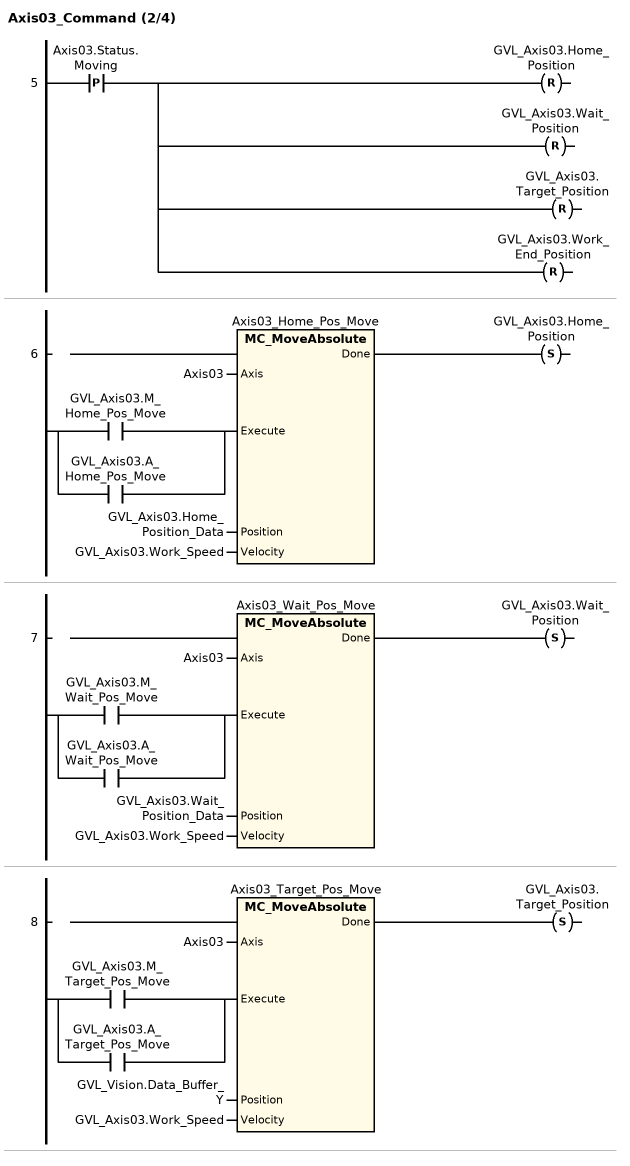
// NETWORK 5
_rt2(CLK := Axis03.Status.Moving);
GVL_Axis03.Home_Position R= _rt2.Q;
GVL_Axis03.Wait_Position R= _rt2.Q;
GVL_Axis03.Target_Position R= _rt2.Q;
GVL_Axis03.Work_End_Position R= _rt2.Q;

// NETWORK 6
Axis03_Home_Pos_Move(
    Axis := Axis03,
    Execute := GVL_Axis03.M_Home_Pos_Move OR GVL_Axis03.A_Home_Pos_Move,
    Position := GVL_Axis03.Home_Position_Data,
    Velocity := GVL_Axis03.Work_Speed); // MC_MoveAbsolute
GVL_Axis03.Home_Position S= Axis03_Home_Pos_Move.Done;

// NETWORK 7
Axis03_Wait_Pos_Move(
    Axis := Axis03,
    Execute := GVL_Axis03.M_Wait_Pos_Move OR GVL_Axis03.A_Wait_Pos_Move,
    Position := GVL_Axis03.Wait_Position_Data,
    Velocity := GVL_Axis03.Work_Speed); // MC_MoveAbsolute
GVL_Axis03.Wait_Position S= Axis03_Wait_Pos_Move.Done;

// NETWORK 8
Axis03_Target_Pos_Move(
    Axis := Axis03,
    Execute := GVL_Axis03.M_Target_Pos_Move OR GVL_Axis03.A_Target_Pos_Move,
    Position := GVL_Vision.Data_Buffer_Y,
    Velocity := GVL_Axis03.Work_Speed); // MC_MoveAbsolute
GVL_Axis03.Target_Position S= Axis03_Target_Pos_Move.Done;

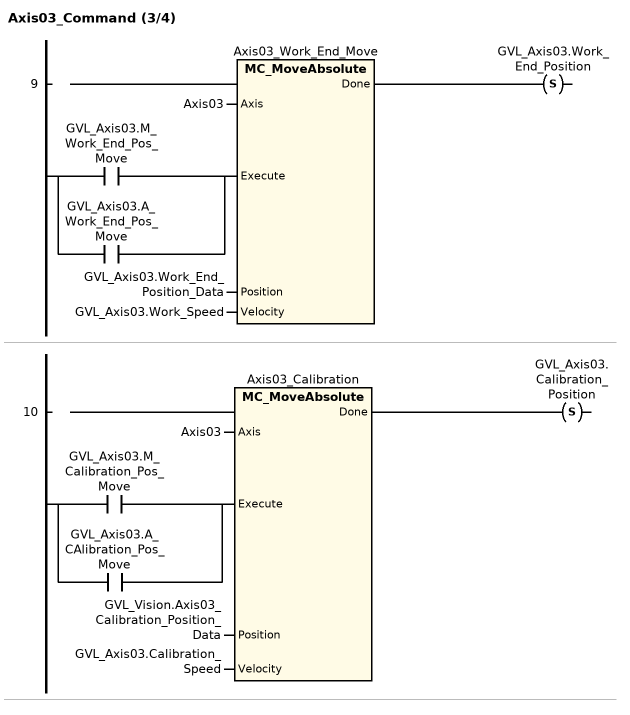
// NETWORK 9
Axis03_Work_End_Move(
    Axis := Axis03,
    Execute := GVL_Axis03.M_Work_End_Pos_Move OR GVL_Axis03.A_Work_End_Pos_Move,
    Position := GVL_Axis03.Work_End_Position_Data,
    Velocity := GVL_Axis03.Work_Speed); // MC_MoveAbsolute
GVL_Axis03.Work_End_Position S= Axis03_Work_End_Move.Done;

// NETWORK 10
Axis03_Calibration(
    Axis := Axis03,
    Execute := GVL_Axis03.M_Calibration_Pos_Move OR GVL_Axis03.A_CAlibration_Pos_Move,
    Position := GVL_Vision.Axis03_Calibration_Position_Data,
    Velocity := GVL_Axis03.Calibration_Speed); // MC_MoveAbsolute
GVL_Axis03.Calibration_Position S= Axis03_Calibration.Done;

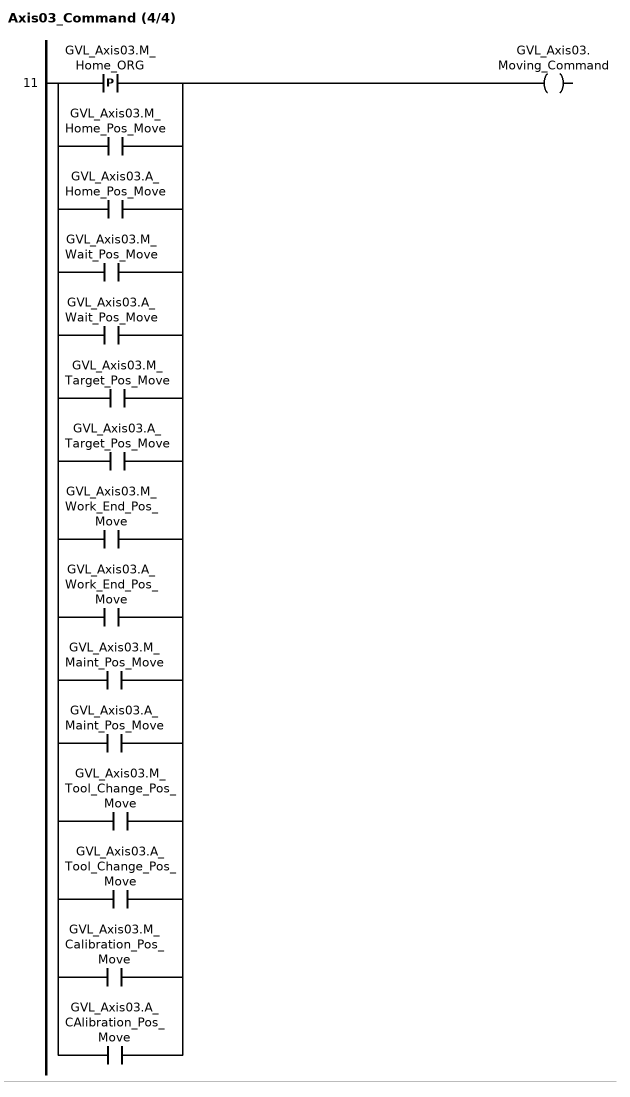
// NETWORK 11
_rt3(CLK := GVL_Axis03.M_Home_ORG);
GVL_Axis03.Moving_Command := _rt3.Q OR GVL_Axis03.M_Home_Pos_Move OR GVL_Axis03.A_Home_Pos_Move OR GVL_Axis03.M_Wait_Pos_Move OR GVL_Axis03.A_Wait_Pos_Move OR GVL_Axis03.M_Target_Pos_Move OR GVL_Axis03.A_Target_Pos_Move OR GVL_Axis03.M_Work_End_Pos_Move OR GVL_Axis03.A_Work_End_Pos_Move OR GVL_Axis03.M_Maint_Pos_Move OR GVL_Axis03.A_Maint_Pos_Move OR GVL_Axis03.M_Tool_Change_Pos_Move OR GVL_Axis03.A_Tool_Change_Pos_Move OR GVL_Axis03.M_Calibration_Pos_Move OR GVL_Axis03.A_CAlibration_Pos_Move;

END_PROGRAM

// ---- POUs/Axis03_Y/Axis03_Manual.TcPOU
PROGRAM Axis03_Manual
VAR
	Always_ON	:	BOOL	:=TRUE	;//상시 ON 
	Always_OFF	:	BOOL	:=FALSE	;//상시 OFF
END_VAR
VAR // added by the converter: edge detectors and wires of the graphical bodies
    _rt1, _rt2, _rt3 : R_TRIG;
END_VAR

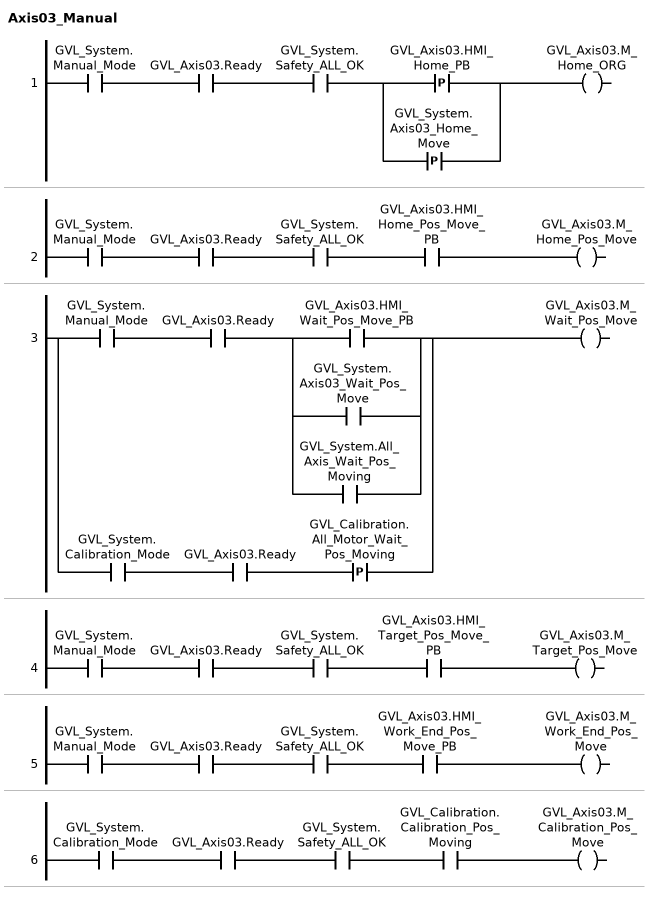
// NETWORK 1
_rt1(CLK := GVL_Axis03.HMI_Home_PB);
_rt2(CLK := GVL_System.Axis03_Home_Move);
GVL_Axis03.M_Home_ORG := GVL_System.Manual_Mode AND GVL_Axis03.Ready AND GVL_System.Safety_ALL_OK AND (_rt1.Q OR _rt2.Q);

// NETWORK 2
GVL_Axis03.M_Home_Pos_Move := GVL_System.Manual_Mode AND GVL_Axis03.Ready AND GVL_System.Safety_ALL_OK AND GVL_Axis03.HMI_Home_Pos_Move_PB;

// NETWORK 3
_rt3(CLK := GVL_Calibration.All_Motor_Wait_Pos_Moving);
GVL_Axis03.M_Wait_Pos_Move := GVL_System.Manual_Mode AND GVL_Axis03.Ready AND (GVL_Axis03.HMI_Wait_Pos_Move_PB OR GVL_System.Axis03_Wait_Pos_Move OR GVL_System.All_Axis_Wait_Pos_Moving) OR GVL_System.Calibration_Mode AND GVL_Axis03.Ready AND _rt3.Q;

// NETWORK 4
GVL_Axis03.M_Target_Pos_Move := GVL_System.Manual_Mode AND GVL_Axis03.Ready AND GVL_System.Safety_ALL_OK AND GVL_Axis03.HMI_Target_Pos_Move_PB;

// NETWORK 5
GVL_Axis03.M_Work_End_Pos_Move := GVL_System.Manual_Mode AND GVL_Axis03.Ready AND GVL_System.Safety_ALL_OK AND GVL_Axis03.HMI_Work_End_Pos_Move_PB;

// NETWORK 6
GVL_Axis03.M_Calibration_Pos_Move := GVL_System.Calibration_Mode AND GVL_Axis03.Ready AND GVL_System.Safety_ALL_OK AND GVL_Calibration.Calibration_Pos_Moving;

END_PROGRAM

// ---- POUs/Axis03_Y/Axis03_Auto.TcPOU
PROGRAM Axis03_Auto
VAR
//System_Bit
	Always_ON	:	BOOL	:=TRUE	;//상시 ON 
	Always_OFF	:	BOOL	:=FALSE	;//상시 OFF
END_VAR

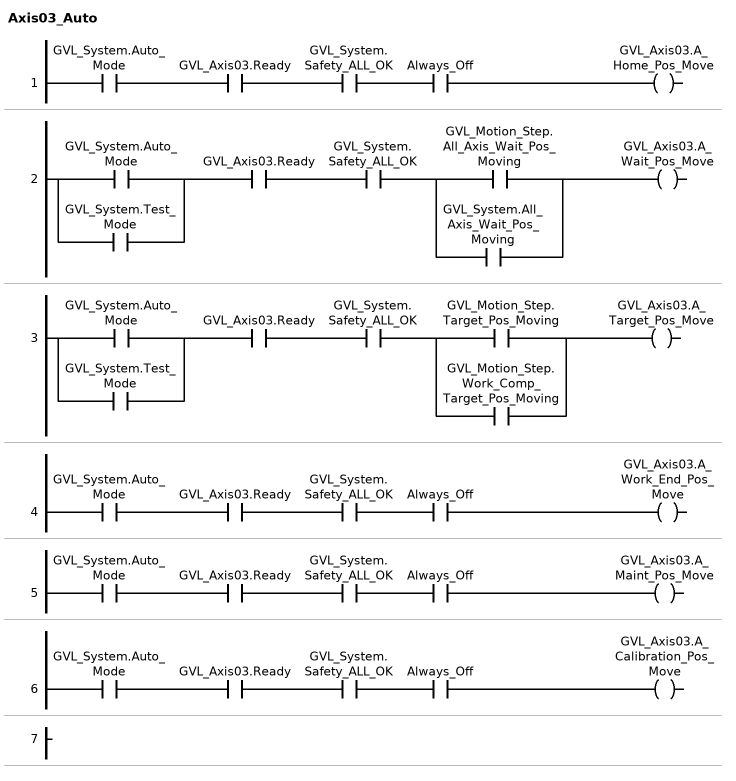
// NETWORK 1
GVL_Axis03.A_Home_Pos_Move := GVL_System.Auto_Mode AND GVL_Axis03.Ready AND GVL_System.Safety_ALL_OK AND Always_Off;

// NETWORK 2
GVL_Axis03.A_Wait_Pos_Move := (GVL_System.Auto_Mode OR GVL_System.Test_Mode) AND GVL_Axis03.Ready AND GVL_System.Safety_ALL_OK AND (GVL_Motion_Step.All_Axis_Wait_Pos_Moving OR GVL_System.All_Axis_Wait_Pos_Moving);

// NETWORK 3
GVL_Axis03.A_Target_Pos_Move := (GVL_System.Auto_Mode OR GVL_System.Test_Mode) AND GVL_Axis03.Ready AND GVL_System.Safety_ALL_OK AND (GVL_Motion_Step.Target_Pos_Moving OR GVL_Motion_Step.Work_Comp_Target_Pos_Moving);

// NETWORK 4
GVL_Axis03.A_Work_End_Pos_Move := GVL_System.Auto_Mode AND GVL_Axis03.Ready AND GVL_System.Safety_ALL_OK AND Always_Off;

// NETWORK 5
GVL_Axis03.A_Maint_Pos_Move := GVL_System.Auto_Mode AND GVL_Axis03.Ready AND GVL_System.Safety_ALL_OK AND Always_Off;

// NETWORK 6
GVL_Axis03.A_Calibration_Pos_Move := GVL_System.Auto_Mode AND GVL_Axis03.Ready AND GVL_System.Safety_ALL_OK AND Always_Off;

// NETWORK 7

END_PROGRAM

// ---- POUs/Axis03_Y/Axis03_Alarm.TcPOU
PROGRAM Axis03_Alarm
VAR
	Always_ON	:	BOOL	:=TRUE	;//상시 ON 
	Always_OFF	:	BOOL	:=FALSE	;//상시 OFF
END_VAR

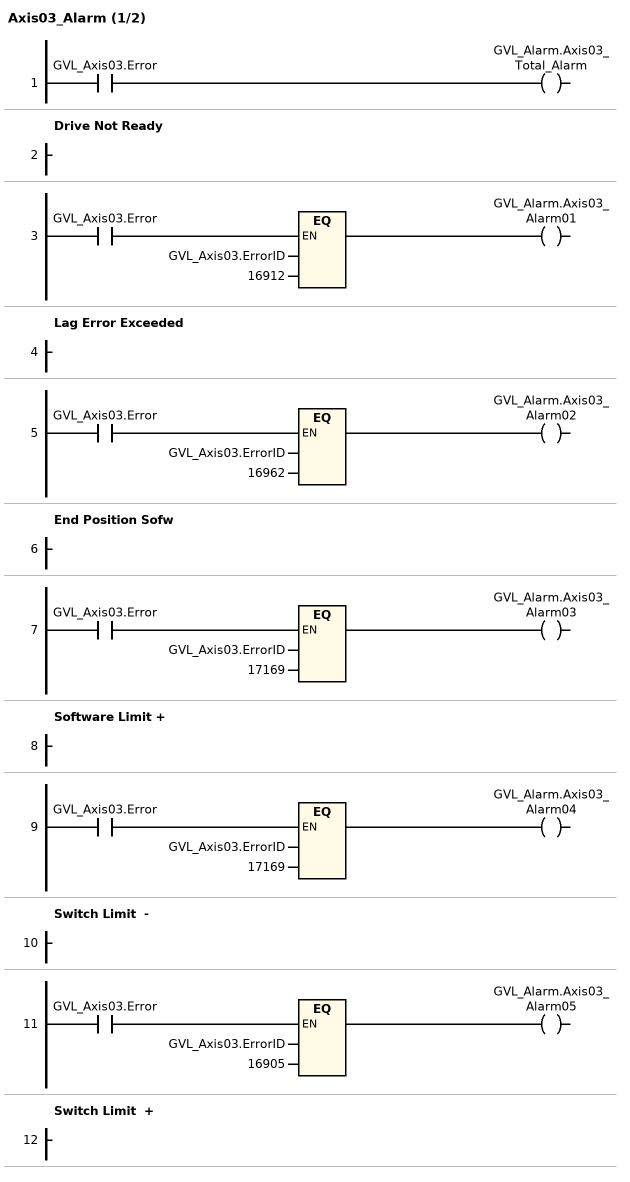
// NETWORK 1
GVL_Alarm.Axis03_Total_Alarm := GVL_Axis03.Error;

// NETWORK 2: Drive Not Ready

// NETWORK 3
GVL_Alarm.Axis03_Alarm01 := GVL_Axis03.Error AND GVL_Axis03.ErrorID = 16912;

// NETWORK 4: Lag Error Exceeded

// NETWORK 5
GVL_Alarm.Axis03_Alarm02 := GVL_Axis03.Error AND GVL_Axis03.ErrorID = 16962;

// NETWORK 6: End Position Sofw

// NETWORK 7
GVL_Alarm.Axis03_Alarm03 := GVL_Axis03.Error AND GVL_Axis03.ErrorID = 17169;

// NETWORK 8: Software Limit +

// NETWORK 9
GVL_Alarm.Axis03_Alarm04 := GVL_Axis03.Error AND GVL_Axis03.ErrorID = 17169;

// NETWORK 10: Switch Limit -

// NETWORK 11
GVL_Alarm.Axis03_Alarm05 := GVL_Axis03.Error AND GVL_Axis03.ErrorID = 16905;

// NETWORK 12: Switch Limit +

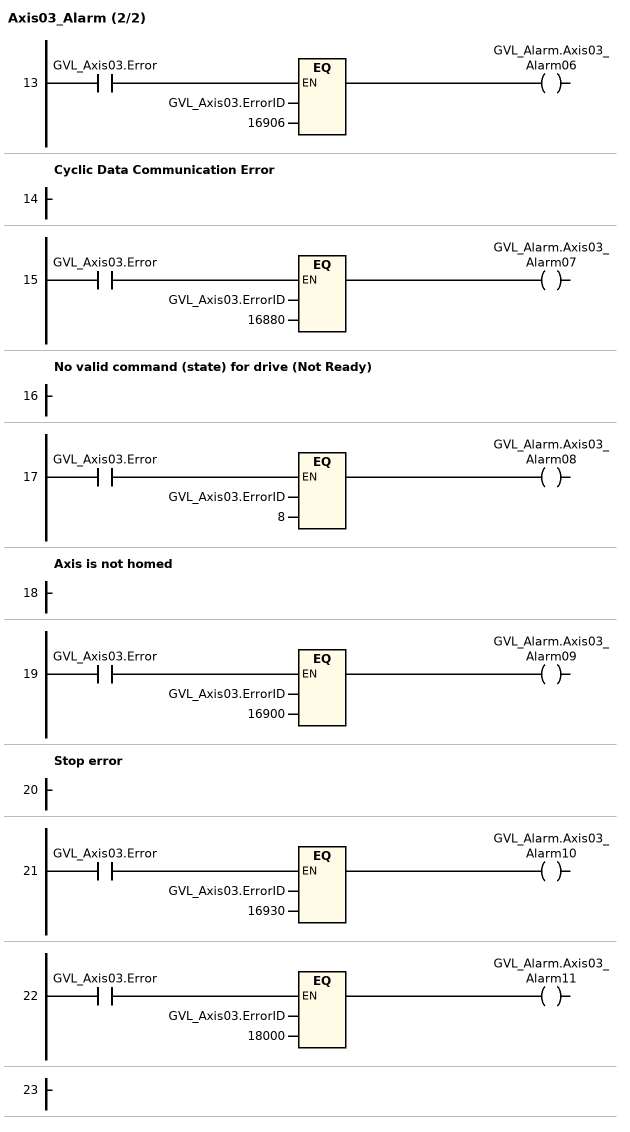
// NETWORK 13
GVL_Alarm.Axis03_Alarm06 := GVL_Axis03.Error AND GVL_Axis03.ErrorID = 16906;

// NETWORK 14: Cyclic Data Communication Error

// NETWORK 15
GVL_Alarm.Axis03_Alarm07 := GVL_Axis03.Error AND GVL_Axis03.ErrorID = 16880;

// NETWORK 16: No valid command (state) for drive (Not Ready)

// NETWORK 17
GVL_Alarm.Axis03_Alarm08 := GVL_Axis03.Error AND GVL_Axis03.ErrorID = 8;

// NETWORK 18: Axis is not homed

// NETWORK 19
GVL_Alarm.Axis03_Alarm09 := GVL_Axis03.Error AND GVL_Axis03.ErrorID = 16900;

// NETWORK 20: Stop error

// NETWORK 21
GVL_Alarm.Axis03_Alarm10 := GVL_Axis03.Error AND GVL_Axis03.ErrorID = 16930;

// NETWORK 22
GVL_Alarm.Axis03_Alarm11 := GVL_Axis03.Error AND GVL_Axis03.ErrorID = 18000;

// NETWORK 23

END_PROGRAM

// ---- POUs/Axis04_Z/Axis04_Status.TcPOU
PROGRAM Axis04_Status
VAR
//System_Bit
	Always_ON	:	BOOL	:=TRUE	;//상시 ON 
	Always_OFF	:	BOOL	:=FALSE	;//상시 OFF
	
//Motor_Command
	Axis04_Status_01: MC_ReadStatus;
	Axis04_Position_Read_01: MC_ReadActualPosition;
	Axis04_Velocity_Read_01: MC_ReadActualVelocity;
	Axis04_Reset_01: MC_Reset;
	Axis04_Stop_01: MC_Stop;
	Torque_Down : UINT := 1500;
	Torque_Up : UINT := 1500;
END_VAR
VAR // added by the converter: edge detectors and wires of the graphical bodies
    _rt1 : R_TRIG;
END_VAR

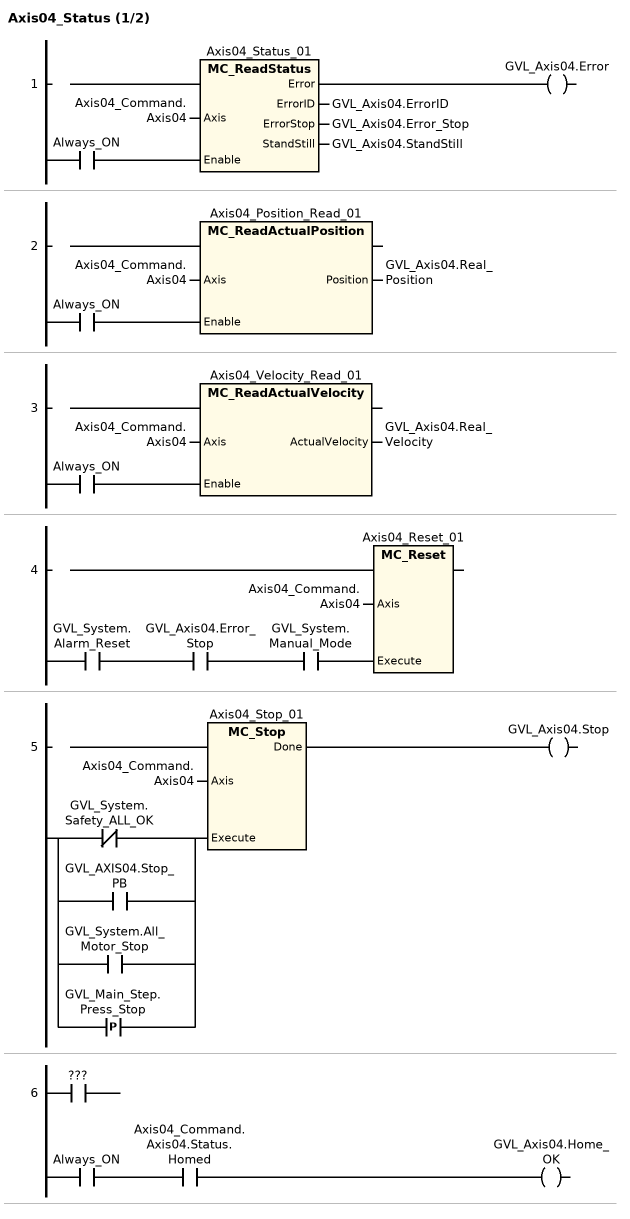
// NETWORK 1
Axis04_Status_01(
    Axis := Axis04_Command.Axis04,
    Enable := Always_ON,
    Error => GVL_Axis04.Error,
    ErrorID => GVL_Axis04.ErrorID,
    ErrorStop => GVL_Axis04.Error_Stop,
    StandStill => GVL_Axis04.StandStill); // MC_ReadStatus

// NETWORK 2
Axis04_Position_Read_01(
    Axis := Axis04_Command.Axis04,
    Enable := Always_ON,
    Position => GVL_Axis04.Real_Position); // MC_ReadActualPosition

// NETWORK 3
Axis04_Velocity_Read_01(
    Axis := Axis04_Command.Axis04,
    Enable := Always_ON,
    ActualVelocity => GVL_Axis04.Real_Velocity); // MC_ReadActualVelocity

// NETWORK 4
Axis04_Reset_01(Axis := Axis04_Command.Axis04, Execute := GVL_System.Alarm_Reset AND GVL_Axis04.Error_Stop AND GVL_System.Manual_Mode); // MC_Reset

// NETWORK 5
_rt1(CLK := GVL_Main_Step.Press_Stop);
Axis04_Stop_01(Axis := Axis04_Command.Axis04, Execute := NOT GVL_System.Safety_ALL_OK OR GVL_AXIS04.Stop_PB OR GVL_System.All_Motor_Stop OR _rt1.Q); // MC_Stop
GVL_Axis04.Stop := Axis04_Stop_01.Done;

// NETWORK 6
GVL_Axis04.Home_OK := Always_ON AND Axis04_Command.Axis04.Status.Homed;

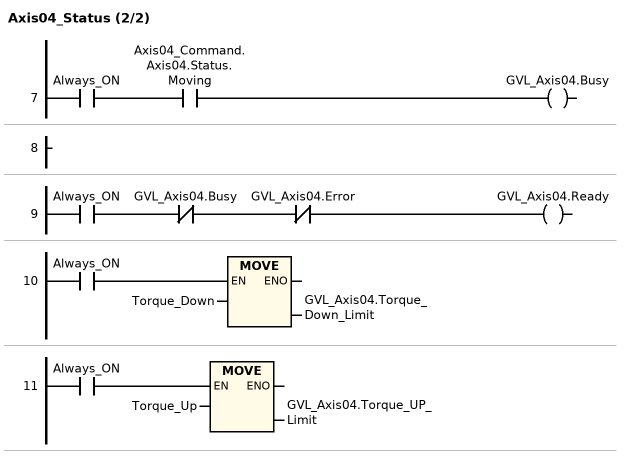
// NETWORK 7
GVL_Axis04.Busy := Always_ON AND Axis04_Command.Axis04.Status.Moving;

// NETWORK 8

// NETWORK 9
GVL_Axis04.Ready := Always_ON AND NOT GVL_Axis04.Busy AND NOT GVL_Axis04.Error;

// NETWORK 10
IF Always_ON THEN GVL_Axis04.Torque_Down_Limit := Torque_Down; END_IF

// NETWORK 11
IF Always_ON THEN GVL_Axis04.Torque_UP_Limit := Torque_Up; END_IF

END_PROGRAM

// ---- POUs/Axis04_Z/Axis04_Command.TcPOU
PROGRAM Axis04_Command
VAR
//SysTem_Bit
	Always_ON	:	BOOL	:=TRUE	;//상시 ON
	Always_OFF	:	BOOL	:=FALSE	;//상시 OFF
//Motor_Command
	Axis04: AXIS_REF;											//회전축
	Axis04_MC_Power: MC_Power;
	Axis04_MC_Home: FB_HomeBeforeMoveAX8000:=(channel:=2);
	Axis04_Jog: MC_Jog;
	Axis04_Home_Pos_Move: MC_MoveAbsolute;
	Axis04_Wait_Pos_Move: MC_MoveAbsolute;
	Axis04_Target_Pos_Move: MC_MoveAbsolute;
	Axis04_Work_End_Move: MC_MoveAbsolute;
	Axis04_Maint_Move: MC_MoveAbsolute;
	Axis04_Tool_Change_Move: MC_MoveAbsolute;
	Axis04_Mastering_Move: MC_MoveAbsolute;	
	
	Axis04_Calibration_Move: MC_MoveAbsolute;
	
	Axis04_Work_Torque: MC_TorqueControl;
	Axis04_Work_Torque2: MC_TorqueControl;
	Options: ST_TorqueControlOptions;
	Timer03: TON;
	Axis04_Cleaning_Pos_Move: MC_MoveAbsolute;
	keb_Z: BOOL;
	Keb_Z_data_PB: BOOL;
END_VAR

VAR_INPUT
	MC_Return_Move: MC_MoveAbsolute;
END_VAR
VAR // added by the converter: edge detectors and wires of the graphical bodies
    _rt1, _rt2 : R_TRIG;
END_VAR

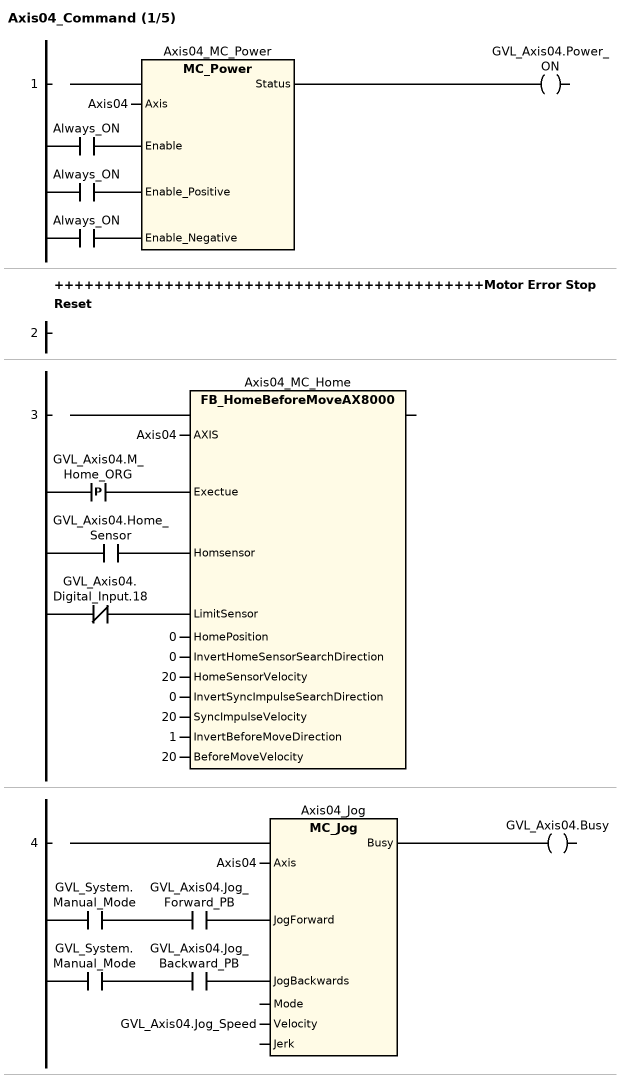
// NETWORK 1
Axis04_MC_Power(
    Axis := Axis04,
    Enable := Always_ON,
    Enable_Positive := Always_ON,
    Enable_Negative := Always_ON); // MC_Power
GVL_Axis04.Power_ON := Axis04_MC_Power.Status;

// NETWORK 2: +++++++++++++++++++++++++++++++++++++++++++Motor Error Stop Reset

// NETWORK 3
_rt1(CLK := GVL_Axis04.M_Home_ORG);
Axis04_MC_Home(
    AXIS := Axis04,
    Exectue := _rt1.Q,
    Homsensor := GVL_Axis04.Home_Sensor,
    LimitSensor := NOT GVL_Axis04.Digital_Input.18,
    HomePosition := 0,
    InvertHomeSensorSearchDirection := 0,
    HomeSensorVelocity := 20,
    InvertSyncImpulseSearchDirection := 0,
    SyncImpulseVelocity := 20,
    InvertBeforeMoveDirection := 1,
    BeforeMoveVelocity := 20); // FB_HomeBeforeMoveAX8000

// NETWORK 4
Axis04_Jog(
    Axis := Axis04,
    JogForward := GVL_System.Manual_Mode AND GVL_Axis04.Jog_Forward_PB,
    JogBackwards := GVL_System.Manual_Mode AND GVL_Axis04.Jog_Backward_PB,
    Velocity := GVL_Axis04.Jog_Speed,
    Busy => GVL_Axis04.Busy); // MC_Jog

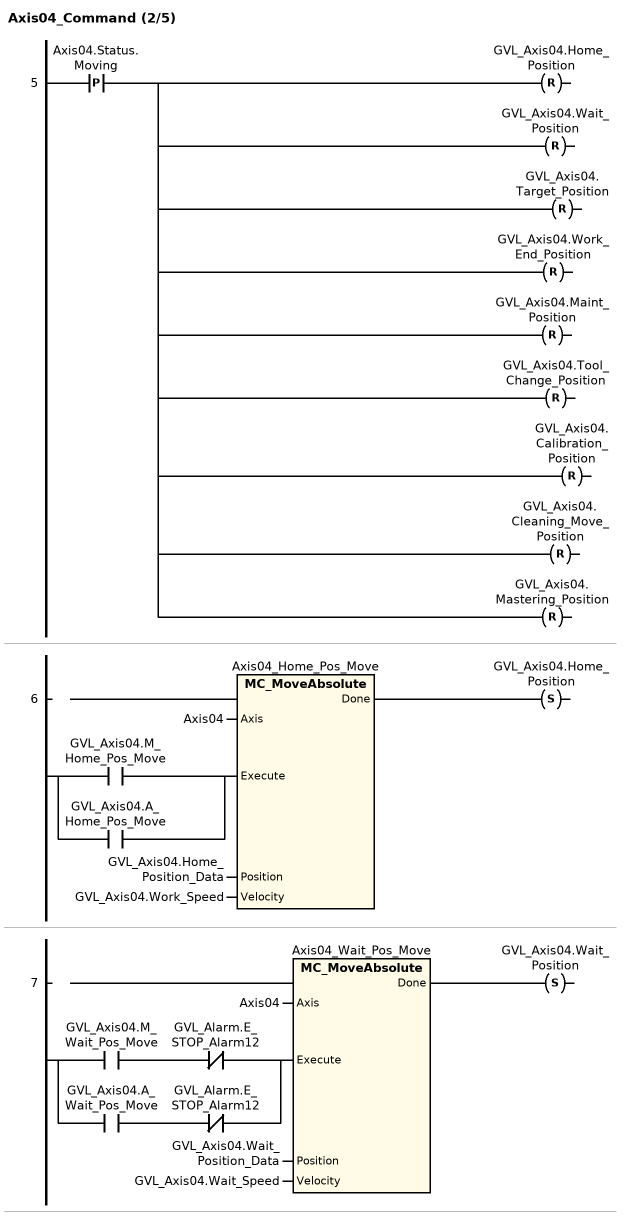
// NETWORK 5
_rt2(CLK := Axis04.Status.Moving);
GVL_Axis04.Home_Position R= _rt2.Q;
GVL_Axis04.Wait_Position R= _rt2.Q;
GVL_Axis04.Target_Position R= _rt2.Q;
GVL_Axis04.Work_End_Position R= _rt2.Q;
GVL_Axis04.Maint_Position R= _rt2.Q;
GVL_Axis04.Tool_Change_Position R= _rt2.Q;
GVL_Axis04.Calibration_Position R= _rt2.Q;
GVL_Axis04.Cleaning_Move_Position R= _rt2.Q;
GVL_Axis04.Mastering_Position R= _rt2.Q;

// NETWORK 6
Axis04_Home_Pos_Move(
    Axis := Axis04,
    Execute := GVL_Axis04.M_Home_Pos_Move OR GVL_Axis04.A_Home_Pos_Move,
    Position := GVL_Axis04.Home_Position_Data,
    Velocity := GVL_Axis04.Work_Speed); // MC_MoveAbsolute
GVL_Axis04.Home_Position S= Axis04_Home_Pos_Move.Done;

// NETWORK 7
Axis04_Wait_Pos_Move(
    Axis := Axis04,
    Execute := GVL_Axis04.M_Wait_Pos_Move AND NOT GVL_Alarm.E_STOP_Alarm12 OR GVL_Axis04.A_Wait_Pos_Move AND NOT GVL_Alarm.E_STOP_Alarm12,
    Position := GVL_Axis04.Wait_Position_Data,
    Velocity := GVL_Axis04.Wait_Speed); // MC_MoveAbsolute
GVL_Axis04.Wait_Position S= Axis04_Wait_Pos_Move.Done;

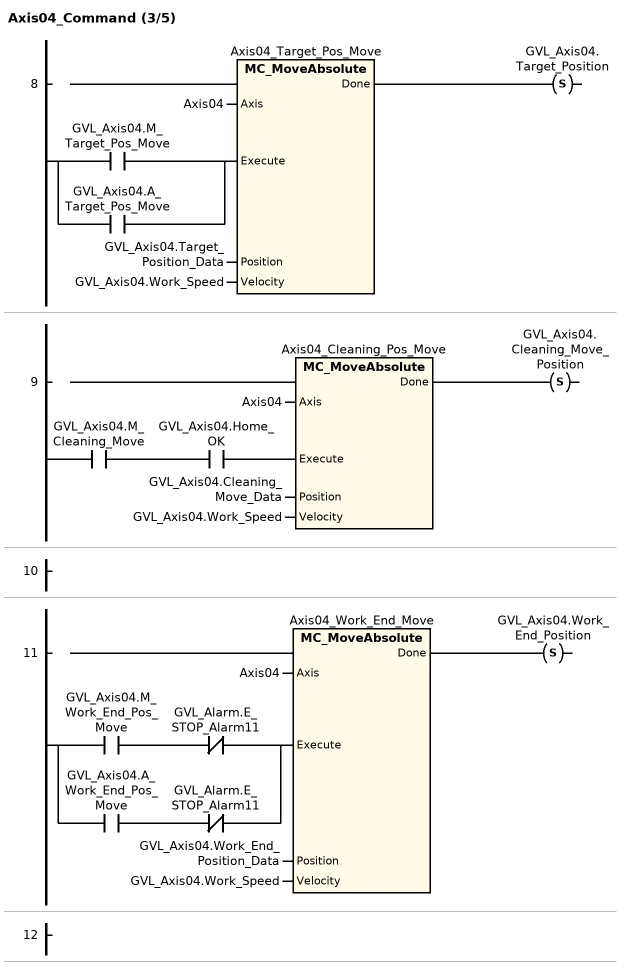
// NETWORK 8
Axis04_Target_Pos_Move(
    Axis := Axis04,
    Execute := GVL_Axis04.M_Target_Pos_Move OR GVL_Axis04.A_Target_Pos_Move,
    Position := GVL_Axis04.Target_Position_Data,
    Velocity := GVL_Axis04.Work_Speed); // MC_MoveAbsolute
GVL_Axis04.Target_Position S= Axis04_Target_Pos_Move.Done;

// NETWORK 9
Axis04_Cleaning_Pos_Move(
    Axis := Axis04,
    Execute := GVL_Axis04.M_Cleaning_Move AND GVL_Axis04.Home_OK,
    Position := GVL_Axis04.Cleaning_Move_Data,
    Velocity := GVL_Axis04.Work_Speed); // MC_MoveAbsolute
GVL_Axis04.Cleaning_Move_Position S= Axis04_Cleaning_Pos_Move.Done;

// NETWORK 10

// NETWORK 11
Axis04_Work_End_Move(
    Axis := Axis04,
    Execute := GVL_Axis04.M_Work_End_Pos_Move AND NOT GVL_Alarm.E_STOP_Alarm11 OR GVL_Axis04.A_Work_End_Pos_Move AND NOT GVL_Alarm.E_STOP_Alarm11,
    Position := GVL_Axis04.Work_End_Position_Data,
    Velocity := GVL_Axis04.Work_Speed); // MC_MoveAbsolute
GVL_Axis04.Work_End_Position S= Axis04_Work_End_Move.Done;

// NETWORK 12

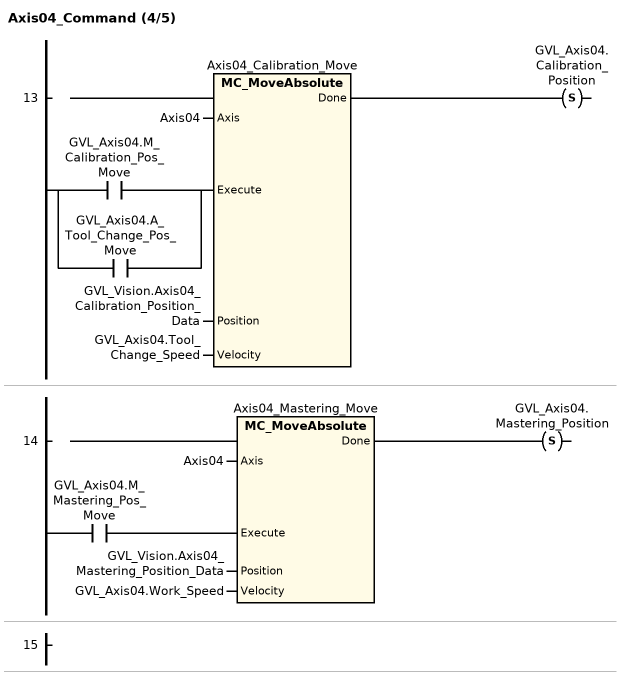
// NETWORK 13
Axis04_Calibration_Move(
    Axis := Axis04,
    Execute := GVL_Axis04.M_Calibration_Pos_Move OR GVL_Axis04.A_Tool_Change_Pos_Move,
    Position := GVL_Vision.Axis04_Calibration_Position_Data,
    Velocity := GVL_Axis04.Tool_Change_Speed); // MC_MoveAbsolute
GVL_Axis04.Calibration_Position S= Axis04_Calibration_Move.Done;

// NETWORK 14
Axis04_Mastering_Move(
    Axis := Axis04,
    Execute := GVL_Axis04.M_Mastering_Pos_Move,
    Position := GVL_Vision.Axis04_Mastering_Position_Data,
    Velocity := GVL_Axis04.Work_Speed); // MC_MoveAbsolute
GVL_Axis04.Mastering_Position S= Axis04_Mastering_Move.Done;

// NETWORK 15

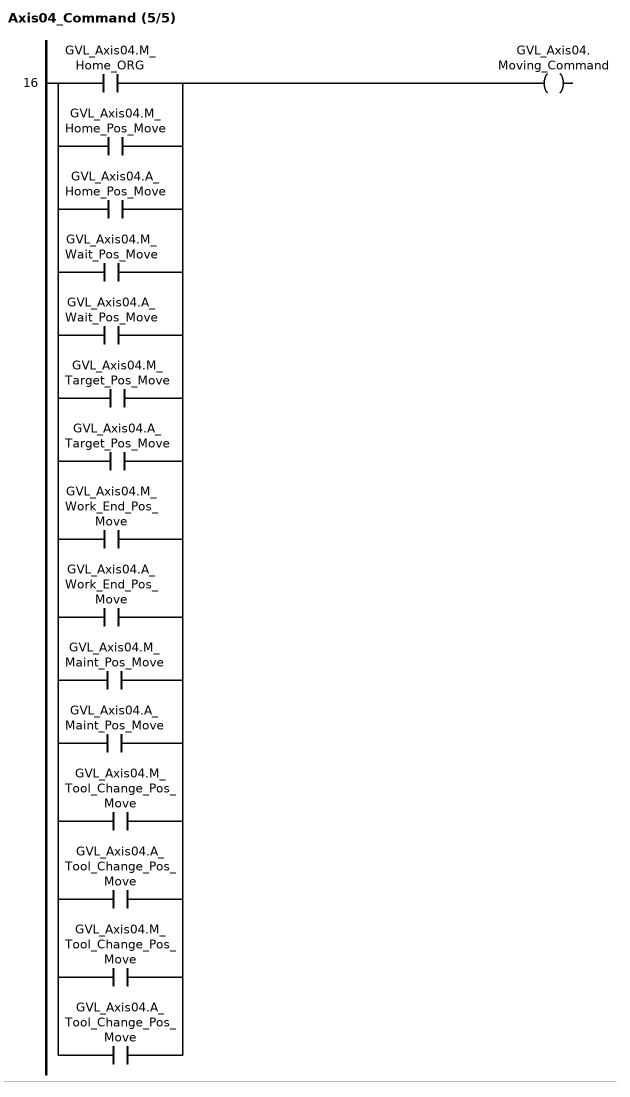
// NETWORK 16
GVL_Axis04.Moving_Command := GVL_Axis04.M_Home_ORG OR GVL_Axis04.M_Home_Pos_Move OR GVL_Axis04.A_Home_Pos_Move OR GVL_Axis04.M_Wait_Pos_Move OR GVL_Axis04.A_Wait_Pos_Move OR GVL_Axis04.M_Target_Pos_Move OR GVL_Axis04.A_Target_Pos_Move OR GVL_Axis04.M_Work_End_Pos_Move OR GVL_Axis04.A_Work_End_Pos_Move OR GVL_Axis04.M_Maint_Pos_Move OR GVL_Axis04.A_Maint_Pos_Move OR GVL_Axis04.M_Tool_Change_Pos_Move OR GVL_Axis04.A_Tool_Change_Pos_Move OR GVL_Axis04.M_Tool_Change_Pos_Move OR GVL_Axis04.A_Tool_Change_Pos_Move;

END_PROGRAM

// ---- POUs/Axis04_Z/Axis04_Manual.TcPOU
PROGRAM Axis04_Manual
VAR
//System_Bit
	Always_ON	:	BOOL	:=TRUE	;//상시 ON 
	Always_OFF	:	BOOL	:=FALSE	;//상시 OFF

END_VAR
VAR // added by the converter: edge detectors and wires of the graphical bodies
    _rt1, _rt2 : R_TRIG;
END_VAR

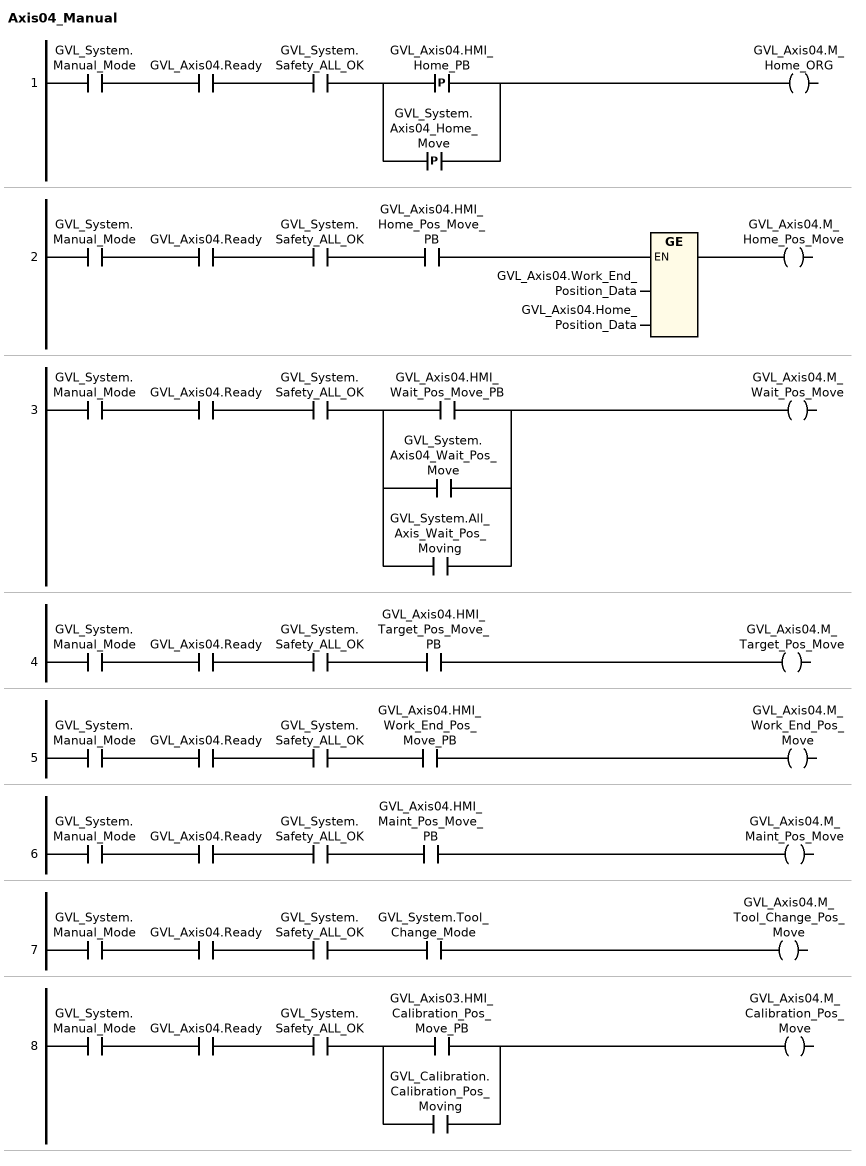
// NETWORK 1
_rt1(CLK := GVL_Axis04.HMI_Home_PB);
_rt2(CLK := GVL_System.Axis04_Home_Move);
GVL_Axis04.M_Home_ORG := GVL_System.Manual_Mode AND GVL_Axis04.Ready AND GVL_System.Safety_ALL_OK AND (_rt1.Q OR _rt2.Q);

// NETWORK 2
GVL_Axis04.M_Home_Pos_Move := GVL_System.Manual_Mode AND GVL_Axis04.Ready AND GVL_System.Safety_ALL_OK AND GVL_Axis04.HMI_Home_Pos_Move_PB AND GVL_Axis04.Work_End_Position_Data >= GVL_Axis04.Home_Position_Data;

// NETWORK 3
GVL_Axis04.M_Wait_Pos_Move := GVL_System.Manual_Mode AND GVL_Axis04.Ready AND GVL_System.Safety_ALL_OK AND (GVL_Axis04.HMI_Wait_Pos_Move_PB OR GVL_System.Axis04_Wait_Pos_Move OR GVL_System.All_Axis_Wait_Pos_Moving);

// NETWORK 4
GVL_Axis04.M_Target_Pos_Move := GVL_System.Manual_Mode AND GVL_Axis04.Ready AND GVL_System.Safety_ALL_OK AND GVL_Axis04.HMI_Target_Pos_Move_PB;

// NETWORK 5
GVL_Axis04.M_Work_End_Pos_Move := GVL_System.Manual_Mode AND GVL_Axis04.Ready AND GVL_System.Safety_ALL_OK AND GVL_Axis04.HMI_Work_End_Pos_Move_PB;

// NETWORK 6
GVL_Axis04.M_Maint_Pos_Move := GVL_System.Manual_Mode AND GVL_Axis04.Ready AND GVL_System.Safety_ALL_OK AND GVL_Axis04.HMI_Maint_Pos_Move_PB;

// NETWORK 7
GVL_Axis04.M_Tool_Change_Pos_Move := GVL_System.Manual_Mode AND GVL_Axis04.Ready AND GVL_System.Safety_ALL_OK AND GVL_System.Tool_Change_Mode;

// NETWORK 8
GVL_Axis04.M_Calibration_Pos_Move := GVL_System.Manual_Mode AND GVL_Axis04.Ready AND GVL_System.Safety_ALL_OK AND (GVL_Axis03.HMI_Calibration_Pos_Move_PB OR GVL_Calibration.Calibration_Pos_Moving);

END_PROGRAM

// ---- POUs/Axis04_Z/Axis04_Auto.TcPOU
PROGRAM Axis04_Auto
VAR
//System_Bit
	Always_ON	:	BOOL	:=TRUE	;//상시 ON 
	Always_OFF	:	BOOL	:=FALSE	;//상시 OFF
END_VAR
VAR // added by the converter: edge detectors and wires of the graphical bodies
    _rt1 : R_TRIG;
END_VAR

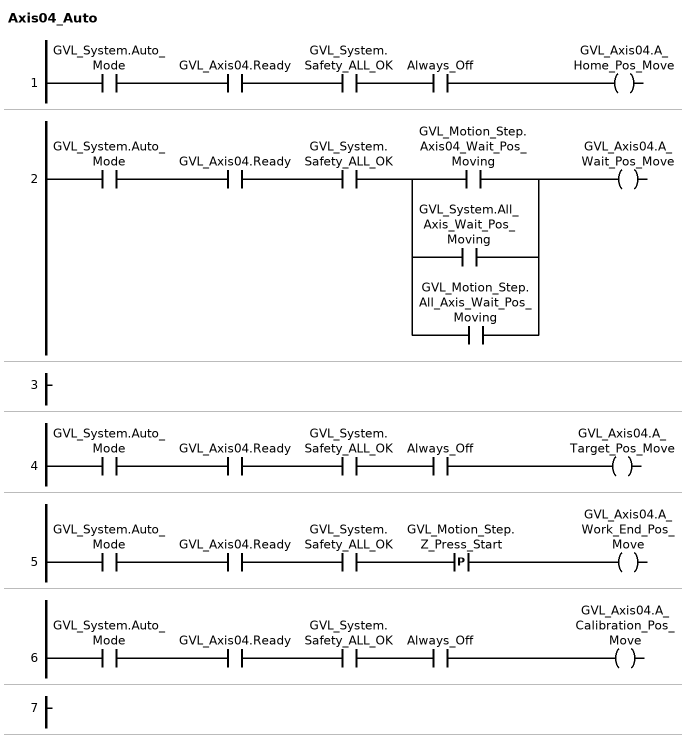
// NETWORK 1
GVL_Axis04.A_Home_Pos_Move := GVL_System.Auto_Mode AND GVL_Axis04.Ready AND GVL_System.Safety_ALL_OK AND Always_Off;

// NETWORK 2
GVL_Axis04.A_Wait_Pos_Move := GVL_System.Auto_Mode AND GVL_Axis04.Ready AND GVL_System.Safety_ALL_OK AND (GVL_Motion_Step.Axis04_Wait_Pos_Moving OR GVL_System.All_Axis_Wait_Pos_Moving OR GVL_Motion_Step.All_Axis_Wait_Pos_Moving);

// NETWORK 3

// NETWORK 4
GVL_Axis04.A_Target_Pos_Move := GVL_System.Auto_Mode AND GVL_Axis04.Ready AND GVL_System.Safety_ALL_OK AND Always_Off;

// NETWORK 5
_rt1(CLK := GVL_Motion_Step.Z_Press_Start);
GVL_Axis04.A_Work_End_Pos_Move := GVL_System.Auto_Mode AND GVL_Axis04.Ready AND GVL_System.Safety_ALL_OK AND _rt1.Q;

// NETWORK 6
GVL_Axis04.A_Calibration_Pos_Move := GVL_System.Auto_Mode AND GVL_Axis04.Ready AND GVL_System.Safety_ALL_OK AND Always_Off;

// NETWORK 7

END_PROGRAM

// ---- POUs/Axis04_Z/Axis04_Alarm.TcPOU
PROGRAM Axis04_Alarm
VAR
//System_Bit
	Always_ON	:	BOOL	:=TRUE	;//상시 ON 
	Always_OFF	:	BOOL	:=FALSE	;//상시 OFF
END_VAR

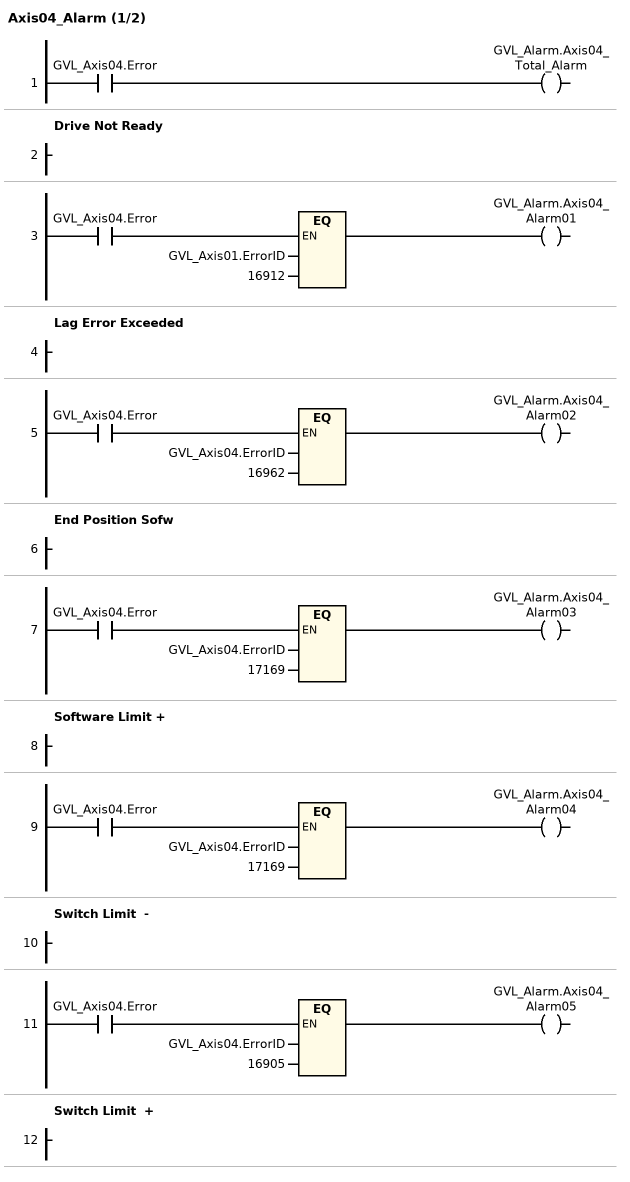
// NETWORK 1
GVL_Alarm.Axis04_Total_Alarm := GVL_Axis04.Error;

// NETWORK 2: Drive Not Ready

// NETWORK 3
GVL_Alarm.Axis04_Alarm01 := GVL_Axis04.Error AND GVL_Axis01.ErrorID = 16912;

// NETWORK 4: Lag Error Exceeded

// NETWORK 5
GVL_Alarm.Axis04_Alarm02 := GVL_Axis04.Error AND GVL_Axis04.ErrorID = 16962;

// NETWORK 6: End Position Sofw

// NETWORK 7
GVL_Alarm.Axis04_Alarm03 := GVL_Axis04.Error AND GVL_Axis04.ErrorID = 17169;

// NETWORK 8: Software Limit +

// NETWORK 9
GVL_Alarm.Axis04_Alarm04 := GVL_Axis04.Error AND GVL_Axis04.ErrorID = 17169;

// NETWORK 10: Switch Limit -

// NETWORK 11
GVL_Alarm.Axis04_Alarm05 := GVL_Axis04.Error AND GVL_Axis04.ErrorID = 16905;

// NETWORK 12: Switch Limit +

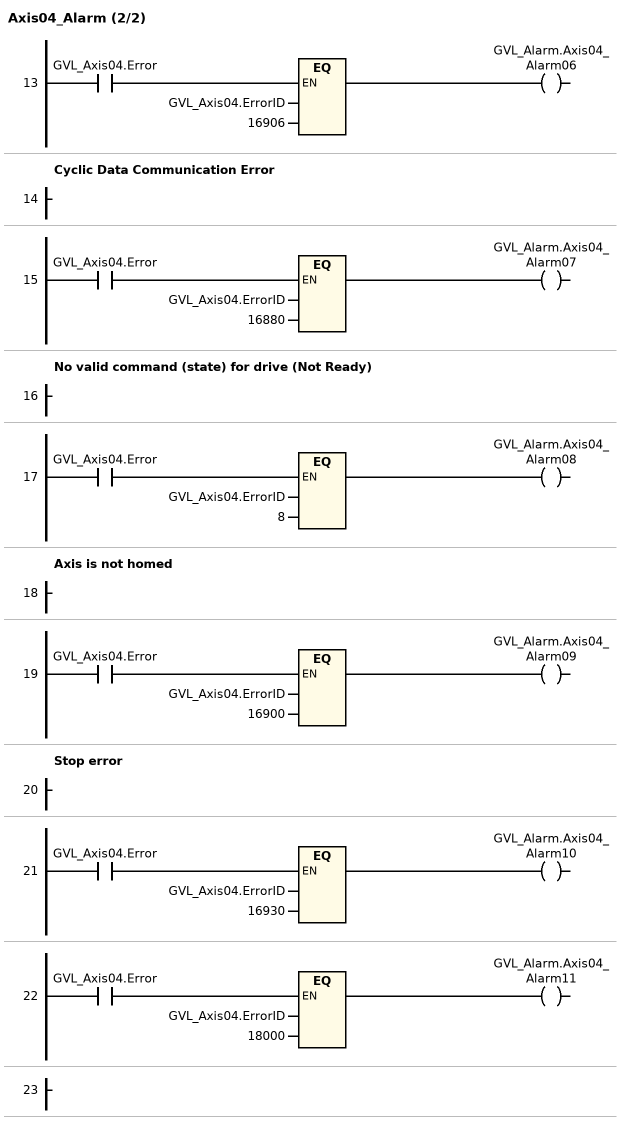
// NETWORK 13
GVL_Alarm.Axis04_Alarm06 := GVL_Axis04.Error AND GVL_Axis04.ErrorID = 16906;

// NETWORK 14: Cyclic Data Communication Error

// NETWORK 15
GVL_Alarm.Axis04_Alarm07 := GVL_Axis04.Error AND GVL_Axis04.ErrorID = 16880;

// NETWORK 16: No valid command (state) for drive (Not Ready)

// NETWORK 17
GVL_Alarm.Axis04_Alarm08 := GVL_Axis04.Error AND GVL_Axis04.ErrorID = 8;

// NETWORK 18: Axis is not homed

// NETWORK 19
GVL_Alarm.Axis04_Alarm09 := GVL_Axis04.Error AND GVL_Axis04.ErrorID = 16900;

// NETWORK 20: Stop error

// NETWORK 21
GVL_Alarm.Axis04_Alarm10 := GVL_Axis04.Error AND GVL_Axis04.ErrorID = 16930;

// NETWORK 22
GVL_Alarm.Axis04_Alarm11 := GVL_Axis04.Error AND GVL_Axis04.ErrorID = 18000;

// NETWORK 23

END_PROGRAM

// ---- POUs/Axis05_Encoder/Axis05_Status.TcPOU
PROGRAM Axis05_Status
VAR
//System_Bit
	Always_ON	:	BOOL	:=TRUE	;//상시 ON 
	Always_OFF	:	BOOL	:=FALSE	;//상시 OFF
	
	Real_Position_Data : ARRAY[0..39999] OF LREAL; // 40,000개 데이터 저장 (2초 보장)
    nIndex          : DINT := 0;                // 배열 인덱스 (0 ~ 39999)

	Axis05_Position_Read: MC_ReadActualPosition;
	Axis05_Velocity_Read: MC_ReadActualVelocity;
	nCounter: INT;
	i: INT;
	Test04: BOOL;
	Test05: BOOL;
	TEST005: BOOL;
	Axis05_Reset_01: MC_Reset;
	
	Set_Pos : MC_SetPosition;
END_VAR

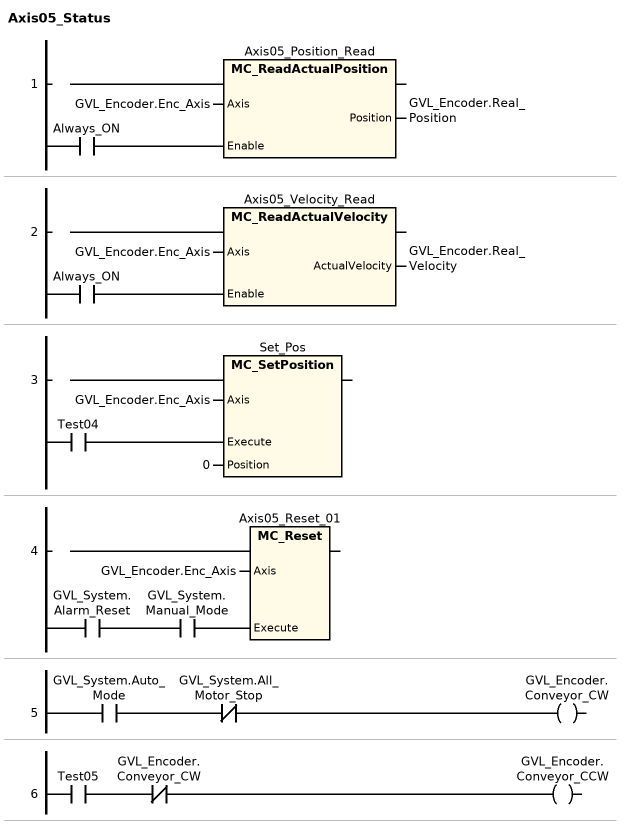
// NETWORK 1
Axis05_Position_Read(
    Axis := GVL_Encoder.Enc_Axis,
    Enable := Always_ON,
    Position => GVL_Encoder.Real_Position); // MC_ReadActualPosition

// NETWORK 2
Axis05_Velocity_Read(
    Axis := GVL_Encoder.Enc_Axis,
    Enable := Always_ON,
    ActualVelocity => GVL_Encoder.Real_Velocity); // MC_ReadActualVelocity

// NETWORK 3
Set_Pos(Axis := GVL_Encoder.Enc_Axis, Execute := Test04, Position := 0); // MC_SetPosition

// NETWORK 4
Axis05_Reset_01(Axis := GVL_Encoder.Enc_Axis, Execute := GVL_System.Alarm_Reset AND GVL_System.Manual_Mode); // MC_Reset

// NETWORK 5
GVL_Encoder.Conveyor_CW := GVL_System.Auto_Mode AND NOT GVL_System.All_Motor_Stop;

// NETWORK 6
GVL_Encoder.Conveyor_CCW := Test05 AND NOT GVL_Encoder.Conveyor_CW;

END_PROGRAM

// ---- POUs/Conv.TcPOU
PROGRAM Conv
VAR
	Motor_CW : R_TRIG;
	Motor_CCW : R_TRIG;
	Conv_Auto : R_TRIG;
END_VAR

IF NOT GVL_System.EMO_SWitch OR NOT GVL_System.Safety_ALL_OK THEN
	GVL_Conv.Conv_Motor_CW := FALSE;
	GVL_Conv.Conv_Motor_CCW := FALSE;
	GVL_Conv.Conv_Motor_High_Speed := FALSE;
	GVL_Conv.Conv_Motor_Normal_Speed := FALSE;
	GVL_Conv.Conv_Motor_Low_Speed := FALSE;
END_IF

Motor_CW(CLK := GVL_Conv.HMI_Motor_CW);
Motor_CCW(CLK := GVL_Conv.HMI_Motor_CCW);
Conv_Auto(CLK := GVL_Conv.Auto_Mode OR NOT GVL_Conv.Auto_Mode);

IF GVL_Conv.Motor_STOP THEN
	GVL_Conv.Conv_Motor_CW := FALSE;
	GVL_Conv.Conv_Motor_CCW := FALSE;
	GVL_Conv.Conv_Motor_High_Speed := FALSE;
	GVL_Conv.Conv_Motor_Normal_Speed := FALSE;
	GVL_Conv.Conv_Motor_Low_Speed := FALSE;
END_IF

IF Motor_CW.Q THEN
 IF GVL_Conv.Conv_Motor_CW THEN
		
		GVL_Conv.Conv_Motor_CW := FALSE;
		GVL_Conv.HMI_Motor_CW := FALSE;
  ELSE
	  	GVL_Conv.Conv_Motor_CW := TRUE;
		GVL_Conv.HMI_Motor_CW := FALSE;
		GVL_Conv.HMI_Motor_CCW := FALSE;
		GVL_Conv.Conv_Motor_CCW := FALSE;
  END_IF
END_IF	
	
IF Motor_CCW.Q THEN
 IF GVL_Conv.Conv_Motor_CCW THEN
		
		GVL_Conv.Conv_Motor_CCW := FALSE;
		GVL_Conv.HMI_Motor_CCW := FALSE;
  ELSE
	  	GVL_Conv.Conv_Motor_CCW := TRUE;
		GVL_Conv.HMI_Motor_CCW := FALSE;
		GVL_Conv.HMI_Motor_CW := FALSE;
		GVL_Conv.Conv_Motor_CW := FALSE;
  END_IF
END_IF	
	
IF GVL_Conv.Auto_Mode = FALSE THEN
	
	GVL_Conv.Conv_Motor_High_Speed := FALSE;
	GVL_Conv.Conv_Motor_Low_Speed := FALSE;
	GVL_Conv.Conv_Motor_Normal_Speed	:= FALSE;
END_IF
IF Conv_Auto.Q THEN
	GVL_Conv.Conv_Motor_High_Speed := FALSE;
	GVL_Conv.Conv_Motor_Low_Speed := FALSE;
	GVL_Conv.Conv_Motor_Normal_Speed	:= FALSE;
END_IF

IF GVL_Conv.Auto_Mode THEN
	
IF GVL_Conv.HMI_Motor_High_Speed THEN
	GVL_Conv.Conv_Motor_High_Speed := TRUE;
	GVL_Conv.Conv_Motor_Low_Speed := FALSE;
	GVL_Conv.Conv_Motor_Normal_Speed	:= FALSE;
END_IF	
IF GVL_Conv.HMI_Motor_Normal_Speed THEN
	GVL_Conv.Conv_Motor_High_Speed := FALSE;
	GVL_Conv.Conv_Motor_Low_Speed := FALSE;
	GVL_Conv.Conv_Motor_Normal_Speed	:= TRUE;
END_IF	
IF GVL_Conv.HMI_Motor_Low_Speed  THEN
	GVL_Conv.Conv_Motor_High_Speed := FALSE;
	GVL_Conv.Conv_Motor_Low_Speed := TRUE;
	GVL_Conv.Conv_Motor_Normal_Speed	:= FALSE;
END_IF	
	
END_IF

END_PROGRAM

// ---- POUs/Alarm/Alarm_Error.TcPOU
PROGRAM Alarm_Error
VAR
//System_Bit
	Always_ON				:	BOOL	:=TRUE	;//상시 ON
	Always_OFF				:	BOOL	:=FALSE	;//상시 OFF
	Alarm_delay: TON;
	Alarm_delay02: TON;
END_VAR

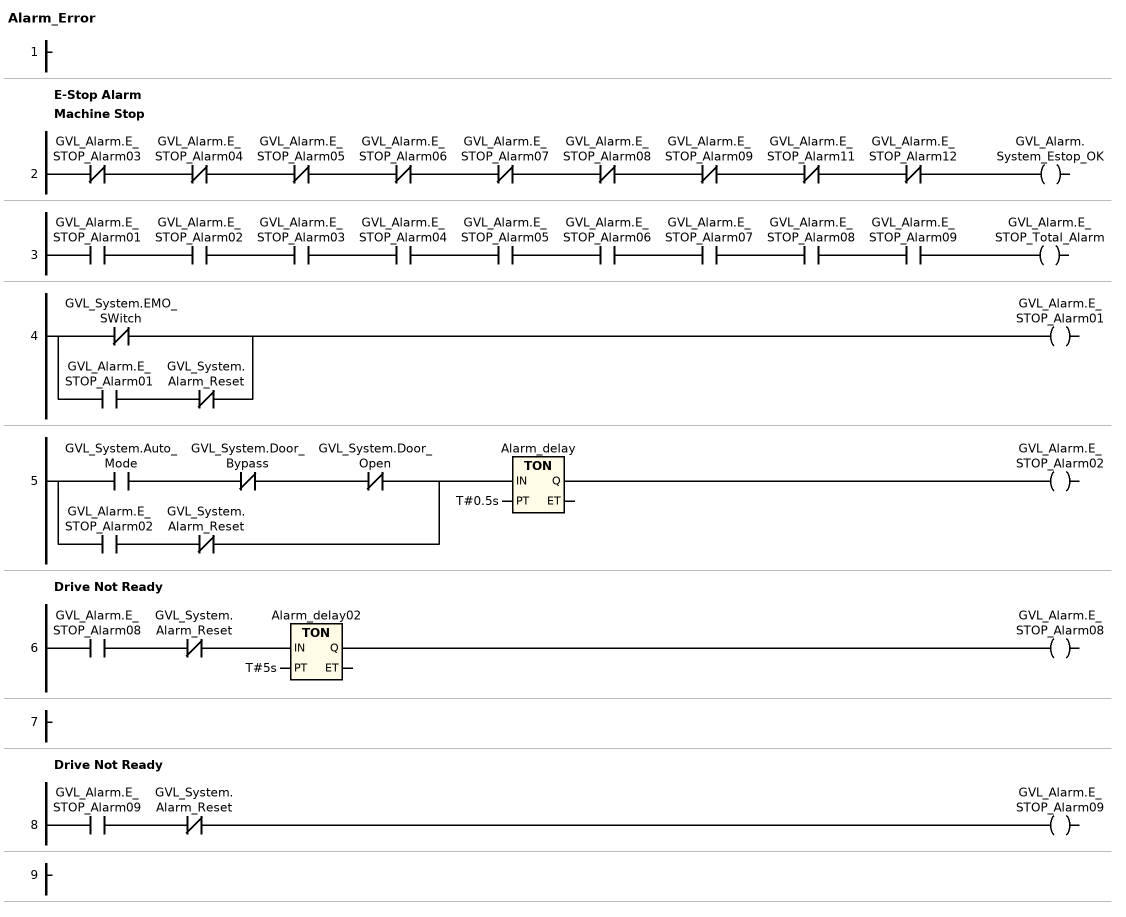
// NETWORK 1

// NETWORK 2: E-Stop Alarm Machine Stop
GVL_Alarm.System_Estop_OK := NOT GVL_Alarm.E_STOP_Alarm03 AND NOT GVL_Alarm.E_STOP_Alarm04 AND NOT GVL_Alarm.E_STOP_Alarm05 AND NOT GVL_Alarm.E_STOP_Alarm06 AND NOT GVL_Alarm.E_STOP_Alarm07 AND NOT GVL_Alarm.E_STOP_Alarm08 AND NOT GVL_Alarm.E_STOP_Alarm09 AND NOT GVL_Alarm.E_STOP_Alarm11 AND NOT GVL_Alarm.E_STOP_Alarm12;

// NETWORK 3
GVL_Alarm.E_STOP_Total_Alarm := GVL_Alarm.E_STOP_Alarm01 AND GVL_Alarm.E_STOP_Alarm02 AND GVL_Alarm.E_STOP_Alarm03 AND GVL_Alarm.E_STOP_Alarm04 AND GVL_Alarm.E_STOP_Alarm05 AND GVL_Alarm.E_STOP_Alarm06 AND GVL_Alarm.E_STOP_Alarm07 AND GVL_Alarm.E_STOP_Alarm08 AND GVL_Alarm.E_STOP_Alarm09;

// NETWORK 4
GVL_Alarm.E_STOP_Alarm01 := NOT GVL_System.EMO_SWitch OR GVL_Alarm.E_STOP_Alarm01 AND NOT GVL_System.Alarm_Reset;

// NETWORK 5
Alarm_delay(IN := GVL_System.Auto_Mode AND NOT GVL_System.Door_Bypass AND NOT GVL_System.Door_Open OR GVL_Alarm.E_STOP_Alarm02 AND NOT GVL_System.Alarm_Reset, PT := T#0.5s); // TON
GVL_Alarm.E_STOP_Alarm02 := Alarm_delay.Q;

// NETWORK 6: Drive Not Ready
Alarm_delay02(IN := GVL_Alarm.E_STOP_Alarm08 AND NOT GVL_System.Alarm_Reset, PT := T#5s); // TON
GVL_Alarm.E_STOP_Alarm08 := Alarm_delay02.Q;

// NETWORK 7

// NETWORK 8: Drive Not Ready
GVL_Alarm.E_STOP_Alarm09 := GVL_Alarm.E_STOP_Alarm09 AND NOT GVL_System.Alarm_Reset;

// NETWORK 9

END_PROGRAM

// ---- POUs/Alarm/Alarm_Warring.TcPOU
PROGRAM Alarm_Warring
VAR
//System_Bit
	Always_ON				:	BOOL	:=TRUE	;//상시 ON
	Always_OFF				:	BOOL	:=FALSE	;//상시 OFF	
END_VAR

// NETWORK 1

// NETWORK 2

END_PROGRAM

// ---- POUs/System/HMI.TcPOU
PROGRAM HMI
VAR
END_VAR

// HMI Start 
IF GVL_HMI.NowScreen_NO = 1 THEN 
	GVL_HMI.ChangeScreen_NO := 2 ;
END_IF
// 가이드 축
IF NOT GVL_HMI.AXIS01_LAMP AND NOT GVL_HMI.AXIS02_LAMP AND NOT GVL_HMI.AXIS03_LAMP AND NOT GVL_HMI.AXIS04_LAMP THEN
	GVL_HMI.AXIS01_LAMP := 1;
	GVL_HMI.AXIS01 := 1;
END_IF	

IF GVL_System.Alarm_Reset AND GVL_HMI.NowScreen_NO = 7 THEN

		GVL_HMI.ChangeScreen_NO := 2;
	
	
END_IF

IF GVL_System.Alarm_Reset AND  GVL_HMI.NowScreen_NO = 6  THEN

		GVL_HMI.ChangeScreen_NO := 2;
	
	
END_IF

IF GVL_System.Alarm_Reset AND  GVL_HMI.NowScreen_NO = 5 THEN

		GVL_HMI.ChangeScreen_NO := 2;
	
	
END_IF
(*
IF GVL_HMI.NowScreen_NO = 3030 THEN
	 GVL_HMI.AXIS01_LAMP := 1;
	 GVL_HMI.AXIS02_LAMP := 0;
	 GVL_HMI.AXIS03_LAMP := 0;
	 GVL_HMI.AXIS04_LAMP := 0;

	 
END_IF

IF GVL_HMI.NowScreen_NO = 3031 THEN
	 GVL_HMI.AXIS01_LAMP := 0;
	 GVL_HMI.AXIS02_LAMP := 1;
	 GVL_HMI.AXIS03_LAMP := 0;
	 GVL_HMI.AXIS04_LAMP := 0;


END_IF

IF GVL_HMI.NowScreen_NO = 3032 THEN
	 GVL_HMI.AXIS01_LAMP := 0;
	 GVL_HMI.AXIS02_LAMP := 0;
	 GVL_HMI.AXIS03_LAMP := 1;
	 GVL_HMI.AXIS04_LAMP := 0;


	 
END_IF

IF GVL_HMI.NowScreen_NO = 3033 THEN
	 GVL_HMI.AXIS01_LAMP := 0;
	 GVL_HMI.AXIS02_LAMP := 0;
	 GVL_HMI.AXIS03_LAMP := 0;
	 GVL_HMI.AXIS04_LAMP := 1;


END_IF

IF GVL_HMI.NowScreen_NO = 3034 THEN
	 GVL_HMI.AXIS01_LAMP := 0;
	 GVL_HMI.AXIS02_LAMP := 0;
	 GVL_HMI.AXIS03_LAMP := 0;
	 GVL_HMI.AXIS04_LAMP := 0;


END_IF

*)

END_PROGRAM

// ---- POUs/System/HOME_MOVE.TcPOU
PROGRAM HOME_MOVE
VAR
	DATA1: LREAL;
	DATAPLS : R_TRIG;
	Manual_TRIG : R_TRIG;
	AUTO_TRIG : R_TRIG;
	WaitMove_TON : TON;		// 대기위치 이동 워치독(도달 실패 시 플래그 강제 해제)
	HomeMove_TON : TON;		// 원점 시퀀스 워치독(완료 실패 시 체인 플래그 강제 해제)
END_VAR
//원점 순서
//1. Z축 잡고 
//2. Z축 올리고
//3.Y축 잡고
//4.Y축 WAIT 포지션
//5. X 축 잡고
//6. 모두 원점 잡으면 올 WAIT 포지션

Manual_TRIG(CLK := GVL_System.Manual_Mode);
AUTO_TRIG(CLK := GVL_System.AUTO_Mode);
IF (GVL_SYSTEM.ALL_Home_Move_PB OR AUTO_TRIG.Q) AND GVL_System.ALL_Motor_Homed AND NOT GVL_System.ALL_Wait_Position THEN
	GVL_System.All_Axis_Wait_Pos_Moving :=TRUE;
	GVL_Axis04.M_Cleaning_Move := FALSE;
END_IF
IF GVL_System.ALL_Wait_Position THEN
	GVL_System.All_Axis_Wait_Pos_Moving :=FALSE;
END_IF
IF Manual_TRIG.Q AND GVL_System.ALL_Motor_Homed THEN
	GVL_Axis04.M_Cleaning_Move := TRUE;
	
END_IF

IF GVL_Axis04.Cleaning_Move_Position THEN
	GVL_Axis04.M_Cleaning_Move := FALSE;
END_IF

IF	(GVL_AxIS02.Wait_Position = TRUE) AND	(GVL_AxIS03.Wait_Position = TRUE) AND	(GVL_AxIS04.Wait_Position = TRUE) AND (GVL_AxIS01.Wait_Position = TRUE) THEN
	
		GVL_System.ALL_Wait_Position := TRUE;
	
ELSE
		GVL_System.ALL_Wait_Position := FALSE;
	
END_IF


IF GVL_SYSTEM.ALL_Home_Move_PB = TRUE AND GVL_System.Manual_Mode = TRUE  AND (GVL_System.ALL_Motor_Homed = FALSE) THEN
	
	GVL_SYSTEM.ALL_Home_Move_Start := TRUE;		// 원점 시작
		
END_IF

IF	(GVL_System.ALL_Home_Move_Start = TRUE) THEN
	
	GVL_System.Axis04_Home_Move := TRUE;	// Z축 원점 시작
	
	IF (GVL_Axis04.Home_OK = TRUE) THEN
		
		GVL_System.Axis02_Home_Move := TRUE;	     //Z축 원점 확인 후 X축 원점 시작  //
		
	END_IF
	IF (GVL_Axis02.Home_OK = TRUE) THEN
		
		GVL_System.Axis03_Home_Move := TRUE;	//   X축 원점 확인 후 가이드 Y,R 축 모두 원점 시작 GVL_System.Axis04_Home_Move
		
	END_IF
	IF (GVL_Axis03.Home_OK = TRUE) THEN
		GVL_System.Axis01_Home_Move := TRUE;
	END_IF
	
		

	IF	(GVL_System.ALL_Motor_Homed = TRUE) AND (GVL_Axis01.Home_OK = TRUE)  THEN
		//모든 측 원점 확인 후 리셋 및 wait 포지션 이동
		
		GVL_SYSTEM.Axis02_Home_Move := FALSE;
		GVL_SYSTEM.Axis03_Home_Move := FALSE;
		GVL_SYSTEM.Axis04_Home_Move := FALSE;
		GVL_SYSTEM.Axis01_Home_Move := FALSE;
		
		GVL_SYSTEM.Axis02_Wait_Pos_Move := TRUE;
		GVL_SYSTEM.Axis03_Wait_Pos_Move := TRUE;
		GVL_SYSTEM.Axis04_Wait_Pos_Move := TRUE;
		GVL_SYSTEM.Axis01_Wait_Pos_Move := TRUE;
	
	END_IF
	IF	(GVL_System.ALL_Wait_Position = TRUE) THEN
		
		GVL_SYSTEM.ALL_Home_Move_Start 	:= FALSE;
		GVL_SYSTEM.Axis02_Wait_Pos_Move := FALSE;
		GVL_SYSTEM.Axis03_Wait_Pos_Move := FALSE;
		GVL_SYSTEM.Axis04_Wait_Pos_Move := FALSE;
		GVL_SYSTEM.Axis01_Wait_Pos_Move := FALSE;
	END_IF

END_IF

IF GVL_System.All_Initial AND NOT GVL_System.ALL_Motor_Homed THEN
	GVL_SYSTEM.Axis02_Home_Move := FALSE;
	GVL_SYSTEM.Axis03_Home_Move := FALSE;
	GVL_SYSTEM.Axis04_Home_Move := FALSE;
	GVL_SYSTEM.Axis01_Home_Move := FALSE;
	GVL_SYSTEM.ALL_Home_Move_Start := FALSE;
END_IF

// --- 대기위치 이동 워치독 ---
// 해제 조건이 ALL_Wait_Position 뿐이라, 한 축이라도 대기위치 판정에 못 들어가면
// All_Axis_Wait_Pos_Moving/Axis0X_Wait_Pos_Move 가 영구 잔류 → Manual 의
// M_Wait_Pos_Move 가 계속 유지되는 데드락(jog 후 자동 복귀, 완료 불가)이 됐다.
// 20초 내 도달 실패 또는 수동 모드 전환 시 대기이동 요청을 전부 강제 해제한다.
WaitMove_TON(IN := GVL_System.All_Axis_Wait_Pos_Moving
	OR GVL_System.Axis01_Wait_Pos_Move OR GVL_System.Axis02_Wait_Pos_Move
	OR GVL_System.Axis03_Wait_Pos_Move OR GVL_System.Axis04_Wait_Pos_Move,
	PT := T#20S);
IF WaitMove_TON.Q OR Manual_TRIG.Q THEN
	GVL_System.All_Axis_Wait_Pos_Moving := FALSE;
	GVL_System.Axis01_Wait_Pos_Move := FALSE;
	GVL_System.Axis02_Wait_Pos_Move := FALSE;
	GVL_System.Axis03_Wait_Pos_Move := FALSE;
	GVL_System.Axis04_Wait_Pos_Move := FALSE;
	GVL_System.ALL_Home_Move_Start := FALSE;
END_IF

// --- 원점 시퀀스 워치독 ---
// Axis0X_Home_Move 의 해제 조건이 "전축 원점 완료"뿐이라, 한 축이라도 원점 실패
// (jog 가로채기·센서 불량 등)하면 체인 비트가 영구 잔류 → M_Home_ORG 를 계속
// 붙잡아 재시도 불가/영구 미완료가 됐다. 120초 내 완료 실패 또는 오토 모드 전환
// 시 원점 체인을 전부 강제 해제한다. (해제 후 원점 버튼으로 처음부터 재시작)
HomeMove_TON(IN := GVL_System.ALL_Home_Move_Start, PT := T#120S);
IF HomeMove_TON.Q OR AUTO_TRIG.Q THEN
	GVL_SYSTEM.Axis01_Home_Move := FALSE;
	GVL_SYSTEM.Axis02_Home_Move := FALSE;
	GVL_SYSTEM.Axis03_Home_Move := FALSE;
	GVL_SYSTEM.Axis04_Home_Move := FALSE;
	GVL_SYSTEM.ALL_Home_Move_Start := FALSE;
END_IF

END_PROGRAM

// ---- POUs/System/Initial.TcPOU
PROGRAM Initial
VAR
END_VAR

IF  GVL_System.All_Initial AND GVL_System.Manual_Mode THEN
	GVL_Vision.Data_Read_X					:=	0;
	GVL_Vision.Data_Read_Y					:=	0;
	GVL_Vision.Data_Read_R					:=	0;
	GVL_Vision.Data_Buffer_X				:=	0;
	GVL_Vision.Data_Buffer_Y				:=	0;
	GVL_Vision.Data_Buffer_R				:=	0;
	GVL_Vision.Vision_OK					:=	0;
	GVL_Vision.Data_Read_OK					:=	0;
	GVL_Vision.Data_Read_NG					:=	0;
	GVL_Vision.Target_X_Real_Position_Data	:=	0;
	GVL_Axis02.Work_Offset					:=	0;
	GVL_Main_Step.NO 						:=	0;
	GVL_Motion_Step.No						:=	0;
	GVL_Vision.Data_Check					:=	0;
	GVL_Vision.Vision_OK					:= FALSE;
	GVL_Axis04.M_Cleaning_Move := FALSE;
	GVL_Vision.Cam_Trigger := FALSE;
	GVL_Axis04.M_Mastering_Pos_Move := FALSE;
	

	// 원점 이동중/대기위치 이동중 상태 강제 해제 — 초기화 버튼으로 탈출 가능하게
	GVL_System.ALL_Home_Move_Start		:= FALSE;
	GVL_System.Axis01_Home_Move			:= FALSE;
	GVL_System.Axis02_Home_Move			:= FALSE;
	GVL_System.Axis03_Home_Move			:= FALSE;
	GVL_System.Axis04_Home_Move			:= FALSE;
	GVL_System.All_Axis_Wait_Pos_Moving	:= FALSE;
	GVL_System.Axis01_Wait_Pos_Move		:= FALSE;
	GVL_System.Axis02_Wait_Pos_Move		:= FALSE;
	GVL_System.Axis03_Wait_Pos_Move		:= FALSE;
	GVL_System.Axis04_Wait_Pos_Move		:= FALSE;
	GVL_Calibration.Calibration_Pos_Moving := FALSE;
	GVL_Calibration.Motor_Move := FALSE;

END_IF

END_PROGRAM

// ---- POUs/System/System.TcPOU
PROGRAM System
VAR

	
	Always_ON					:	BOOL	:=TRUE;	//상시ON
	Always_OFF					:	BOOL	:=FALSE;//상시OFF

	TON_ON  					: 	TON		; 		// 0.1초 ON 타이머 인스턴스
    TON_OFF 					:	TON		; 		// 0.1초 OFF 타이머 인스턴스
	TON2_ON  					: 	TON		; 		// 1초 ON 타이머 인스턴스
    TON2_OFF 					:	TON		;		 // 1초 OFF 타이머 인스턴스
	
	IO_Test						:	BOOL	;
	Lamp_Test_Green				:	BOOL	;
	Lamp_Test_Yellow			:	BOOL	;
	Lamp_Test_Red				:	BOOL	;
	Lamp_Test_Buzzer			:	BOOL	;
	Manual_Ready : BOOL;
	
	Buzzer						:	BOOL	;
	
	Moving_Motor_Wait_Position: BOOL;
	TEST02: INT;
	TEST06: BOOL;
	Axis02_Power_ON: TON;
	Axis03_Power_ON: TON;
	Axis04_Power_ON: TON;
END_VAR
VAR // added by the converter: edge detectors and wires of the graphical bodies
    _w1 : BOOL;
    _rt1, _rt2, _rt3, _rt4, _rt5, _rt6, _rt7 : R_TRIG;
    _ft1, _ft2 : F_TRIG;
END_VAR

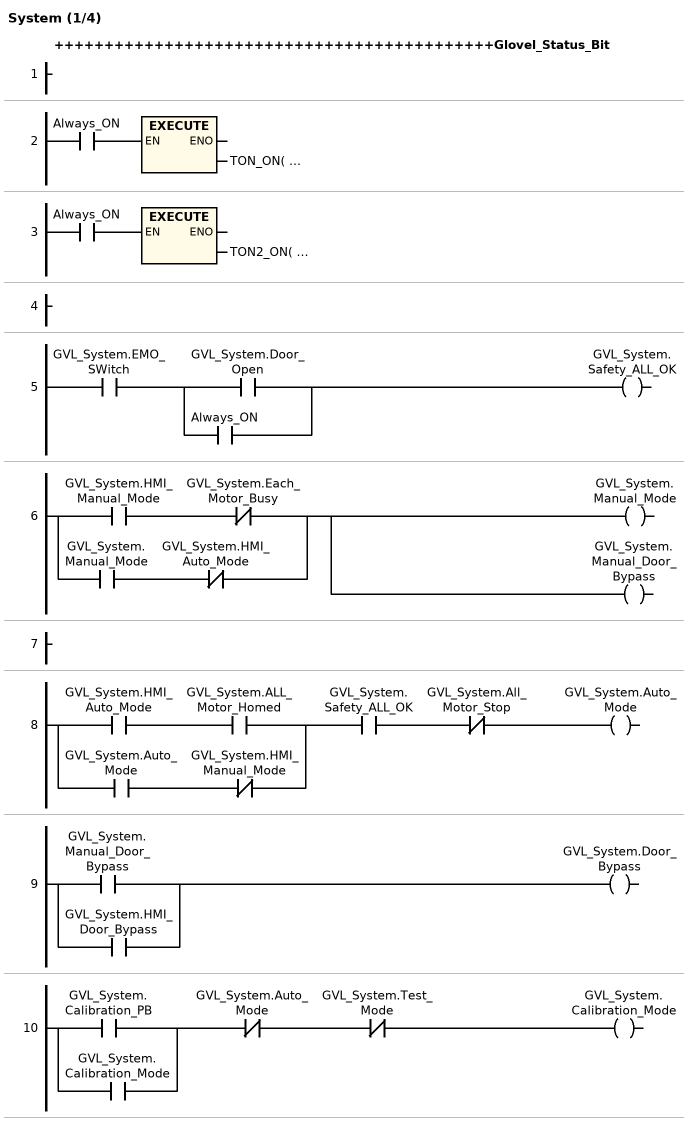
// NETWORK 1: ++++++++++++++++++++++++++++++++++++++++++++Glovel_Status_Bit

// NETWORK 2
IF Always_ON THEN
    TON_ON(
        IN := Always_ON AND NOT TON_OFF.Q,
        PT := T#100ms,
        Q  => 
    );
    
    TON_OFF(
        IN := Always_ON AND TON_ON.Q, 
        PT := T#100ms,
        Q  => 
    );
    
    GVL_System.Pulse_100ms := TON_OFF.IN;
END_IF

// NETWORK 3
IF Always_ON THEN
    TON2_ON(
        IN := Always_ON AND NOT TON2_OFF.Q,
        PT := T#1S,
        Q  => 
    );
    
    TON2_OFF(
        IN := Always_ON AND TON2_ON.Q,
        PT := T#1S,
        Q  => 
    );
    
    GVL_System.Pulse_1S := TON2_OFF.IN;
END_IF

// NETWORK 4

// NETWORK 5
GVL_System.Safety_ALL_OK := GVL_System.EMO_SWitch AND (GVL_System.Door_Open OR Always_ON);

// NETWORK 6
_w1 := GVL_System.HMI_Manual_Mode AND NOT GVL_System.Each_Motor_Busy OR GVL_System.Manual_Mode AND NOT GVL_System.HMI_Auto_Mode;
GVL_System.Manual_Mode := _w1;
GVL_System.Manual_Door_Bypass := _w1;

// NETWORK 7

// NETWORK 8
GVL_System.Auto_Mode := (GVL_System.HMI_Auto_Mode AND GVL_System.ALL_Motor_Homed OR GVL_System.Auto_Mode AND NOT GVL_System.HMI_Manual_Mode) AND GVL_System.Safety_ALL_OK AND NOT GVL_System.All_Motor_Stop;

// NETWORK 9
GVL_System.Door_Bypass := GVL_System.Manual_Door_Bypass OR GVL_System.HMI_Door_Bypass;

// NETWORK 10
GVL_System.Calibration_Mode := (GVL_System.Calibration_PB OR GVL_System.Calibration_Mode) AND NOT GVL_System.Auto_Mode AND NOT GVL_System.Test_Mode;

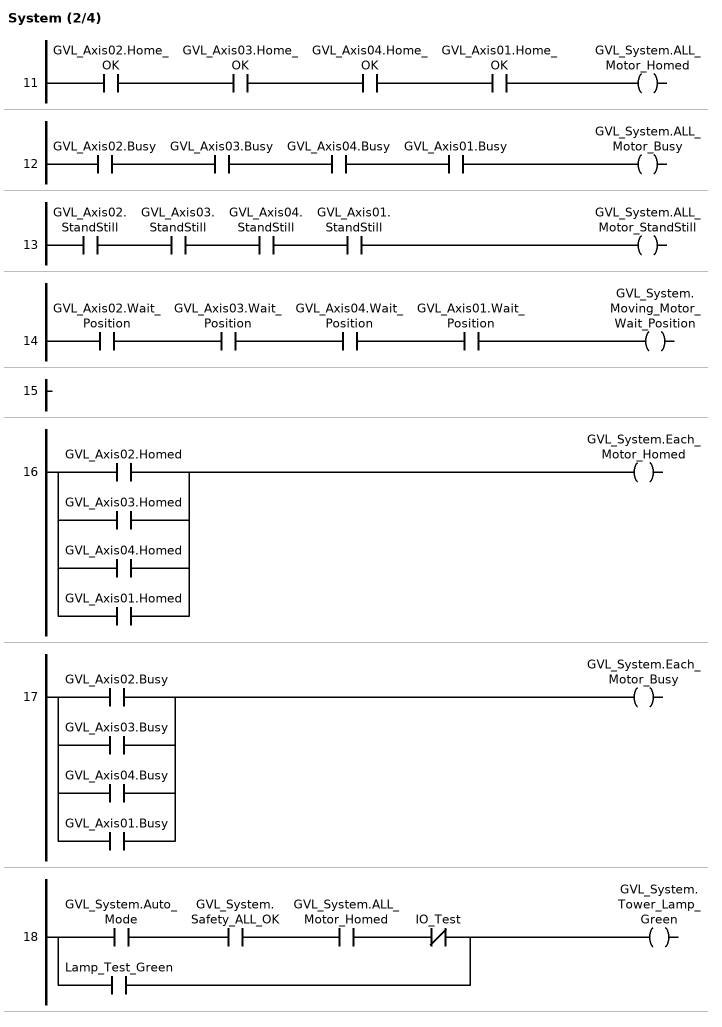
// NETWORK 11
GVL_System.ALL_Motor_Homed := GVL_Axis02.Home_OK AND GVL_Axis03.Home_OK AND GVL_Axis04.Home_OK AND GVL_Axis01.Home_OK;

// NETWORK 12
GVL_System.ALL_Motor_Busy := GVL_Axis02.Busy AND GVL_Axis03.Busy AND GVL_Axis04.Busy AND GVL_Axis01.Busy;

// NETWORK 13
GVL_System.ALL_Motor_StandStill := GVL_Axis02.StandStill AND GVL_Axis03.StandStill AND GVL_Axis04.StandStill AND GVL_Axis01.StandStill;

// NETWORK 14
GVL_System.Moving_Motor_Wait_Position := GVL_Axis02.Wait_Position AND GVL_Axis03.Wait_Position AND GVL_Axis04.Wait_Position AND GVL_Axis01.Wait_Position;

// NETWORK 15

// NETWORK 16
GVL_System.Each_Motor_Homed := GVL_Axis02.Homed OR GVL_Axis03.Homed OR GVL_Axis04.Homed OR GVL_Axis01.Homed;

// NETWORK 17
GVL_System.Each_Motor_Busy := GVL_Axis02.Busy OR GVL_Axis03.Busy OR GVL_Axis04.Busy OR GVL_Axis01.Busy;

// NETWORK 18
GVL_System.Tower_Lamp_Green := GVL_System.Auto_Mode AND GVL_System.Safety_ALL_OK AND GVL_System.ALL_Motor_Homed AND NOT IO_Test OR Lamp_Test_Green;

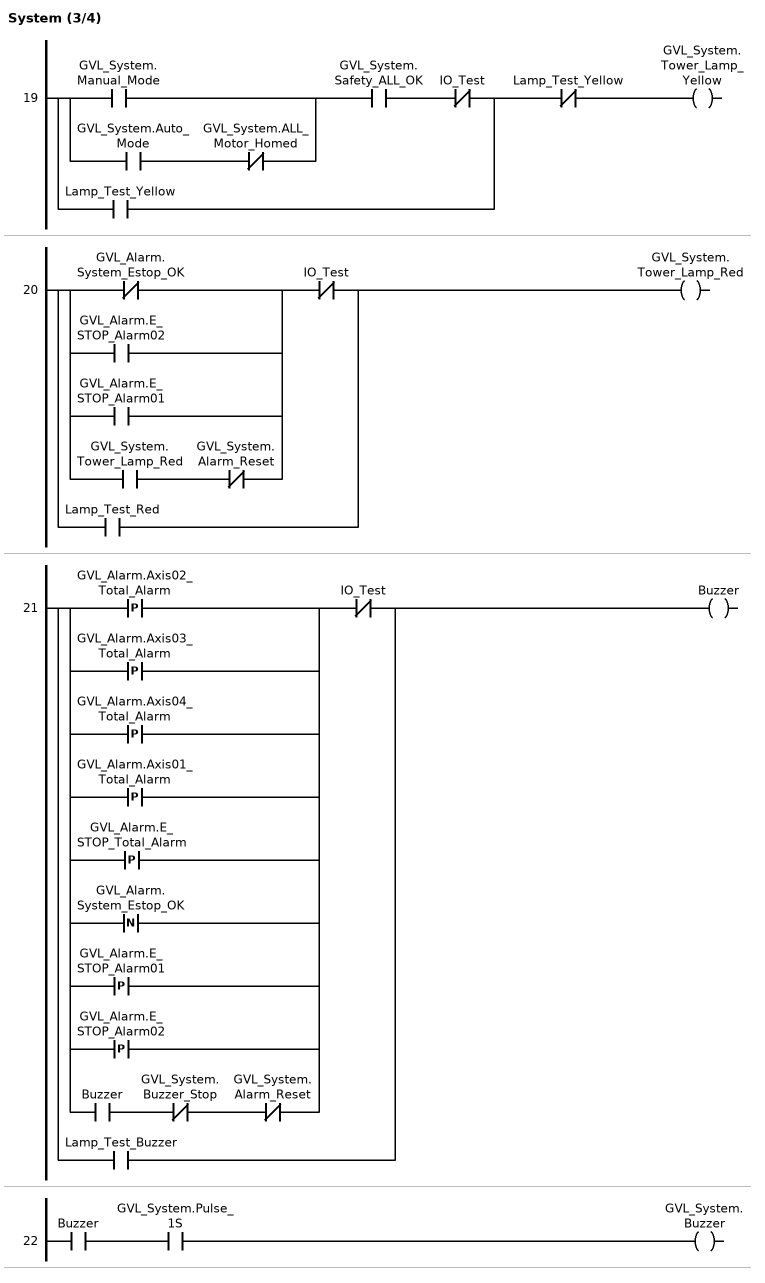
// NETWORK 19
GVL_System.Tower_Lamp_Yellow := ((GVL_System.Manual_Mode OR GVL_System.Auto_Mode AND NOT GVL_System.ALL_Motor_Homed) AND GVL_System.Safety_ALL_OK AND NOT IO_Test OR Lamp_Test_Yellow) AND NOT Lamp_Test_Yellow;

// NETWORK 20
GVL_System.Tower_Lamp_Red := (NOT GVL_Alarm.System_Estop_OK OR GVL_Alarm.E_STOP_Alarm02 OR GVL_Alarm.E_STOP_Alarm01 OR GVL_System.Tower_Lamp_Red AND NOT GVL_System.Alarm_Reset) AND NOT IO_Test OR Lamp_Test_Red;

// NETWORK 21
_rt1(CLK := GVL_Alarm.Axis02_Total_Alarm);
_rt2(CLK := GVL_Alarm.Axis03_Total_Alarm);
_rt3(CLK := GVL_Alarm.Axis04_Total_Alarm);
_rt4(CLK := GVL_Alarm.Axis01_Total_Alarm);
_rt5(CLK := GVL_Alarm.E_STOP_Total_Alarm);
_ft1(CLK := GVL_Alarm.System_Estop_OK);
_rt6(CLK := GVL_Alarm.E_STOP_Alarm01);
_rt7(CLK := GVL_Alarm.E_STOP_Alarm02);
Buzzer := (_rt1.Q OR _rt2.Q OR _rt3.Q OR _rt4.Q OR _rt5.Q OR _ft1.Q OR _rt6.Q OR _rt7.Q OR Buzzer AND NOT GVL_System.Buzzer_Stop AND NOT GVL_System.Alarm_Reset) AND NOT IO_Test OR Lamp_Test_Buzzer;

// NETWORK 22
GVL_System.Buzzer := Buzzer AND GVL_System.Pulse_1S;

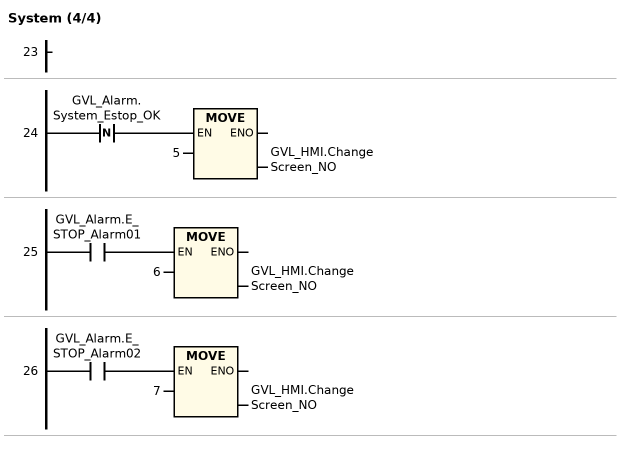
// NETWORK 23

// NETWORK 24
_ft2(CLK := GVL_Alarm.System_Estop_OK);
IF _ft2.Q THEN GVL_HMI.ChangeScreen_NO := 5; END_IF

// NETWORK 25
IF GVL_Alarm.E_STOP_Alarm01 THEN GVL_HMI.ChangeScreen_NO := 6; END_IF

// NETWORK 26
IF GVL_Alarm.E_STOP_Alarm02 THEN GVL_HMI.ChangeScreen_NO := 7; END_IF

END_PROGRAM

// ---- POUs/Vision/Vision_ST.TcPOU
PROGRAM Vision_ST
VAR
    CamTrigger : FB_CamTrigger;   // 캠트리거 파이프라인(센서→트리거, 연속 리얼타임)
END_VAR


// ===== 캠트리거 파이프라인 (파이버 센서 → 카메라 트리거, 연속 리얼타임) =====
CamTrigger(
    Auto_Mode      := GVL_System.Auto_Mode,
    Fiber_Sensor   := GVL_System.Fiber_Sensor,
    Real_Position  := GVL_Encoder.Real_Position,
    Conveyor_CCW   := GVL_Encoder.Conveyor_CCW,
    Trigger_Length := GVL_Vision.Cam_Trigger_Length,
    Reset          := GVL_System.All_Initial);

// 오토모드 캠트리거만 구동 (마스터링은 Mastering.TcPOU 에서 별도 구동, 수동캠트리거 미사용)
IF GVL_System.Auto_Mode THEN GVL_Vision.Cam_Trigger := CamTrigger.Trigger; END_IF

GVL_Vision.Cam_Trig_Position := CamTrigger.Trig_Position;   // Target X 보정 기준(트리거 순간 엔코더)

// ===== Vision Light ON =====
GVL_Vision.Vision_Light_ON := GVL_System.Auto_Mode OR GVL_Vision.Vision_Light_ON;

END_PROGRAM

// ---- POUs/FB_CamTrigger.TcPOU
(* 캠트리거 파이프라인 — 파이버 센서 감지부터 카메라 트리거까지 (연속 리얼타임).
   센서 100ms 디바운스 → 후단(하강엣지)에서 엔코더 기준점을 큐에 push →
   head 기준점 + Trigger_Length 도달 시 1회 트리거 + pop. 오토모드 전용.
   (수동/마스터링 캠트리거는 Mastering.TcPOU 에서 별도 구동)

   pop 안전장치:
     - 큐 만재 시 Push 거부 → Case_Armed 유지(무음 유실 방지)
     - 위치 불연속(엔코더 리셋·대형 역행 점프) 시 큐 flush(stale head 방지)
     - Reset(시스템초기화/사이클말) 시 큐 비움 *)
FUNCTION_BLOCK FB_CamTrigger
VAR_INPUT
    Auto_Mode      : BOOL;     // 오토모드(미오토 시 큐 flush + 트리거 정지)
    Fiber_Sensor   : BOOL;     // 파이버 센서 입력
    Real_Position  : LREAL;    // 엔코더 실제 위치
    Conveyor_CCW   : BOOL;     // 컨베이어 역방향(큐 flush)
    Trigger_Length : LREAL;    // 기준점 + 이 거리 도달 시 트리거(GVL_Vision.Cam_Trigger_Length)
    Reset          : BOOL;     // 시스템초기화/사이클말 큐 비움(레벨, 상승엣지에 1회 clear)
END_VAR
VAR_OUTPUT
    Trigger        : BOOL;     // 0.1s 정형된 캠트리거 펄스(오토 발동분)
    Trig_Position  : LREAL;    // 트리거 순간 엔코더 위치 래치(Target X 보정 기준)
END_VAR
VAR
    Fiber_Trig         : F_TRIG;            // 센서 하강엣지(후단 후보 위치 캡처용)
    Valid_TON          : TON;               // 100ms 연속 ON = 유효 케이스(전단 디바운스)
    Off_TON            : TON;               // 후단 디바운스: OFF_DEBOUNCE 연속 OFF 여야 진짜 후단으로 인정
    Off_Confirm        : R_TRIG;            // 후단 확정(블립 아님) 상승엣지
    Trailing_Pos       : LREAL;             // 하강엣지 순간 캡처한 후단 위치(디바운스 통과 시 이 위치를 push)
    OFF_DEBOUNCE       : TIME := T#50MS;    // 후단 OFF 디바운스 — 부품 간 최소 OFF 보다 짧게 튜닝(길면 가까운 부품 병합)
    Trig_Pulse         : TP;                // 0.1s 펄스 정형
    Reset_Trig         : R_TRIG;            // Reset 상승엣지
    Case_Armed         : BOOL;              // 유효 케이스 무장 → 후단 push 대기, push/flush 시 해제
    bDistReached       : BOOL;              // 이번 스캔 head 가 촬영거리 도달
    Last_Real_Position : LREAL;             // 직전 스캔 엔코더 위치(위치 불연속 감지용)
    Queue              : FB_LRealRingQueue; // 캠트리거 기준점 큐(용량5)
    RESET_JUMP_MIN     : LREAL := 100;      // 역방향 점프 임계(>1스캔 최대 이송) — 엔코더 스케일 맞춰 튜닝
END_VAR

Fiber_Trig(CLK := Fiber_Sensor);
Valid_TON(IN := Fiber_Sensor, PT := T#100MS);
Off_TON(IN := NOT Fiber_Sensor, PT := OFF_DEBOUNCE);   // 후단 디바운스: OFF 가 연속 유지돼야 확정
Off_Confirm(CLK := Off_TON.Q);                          // 확정 후단(블립 아님) 상승엣지
Reset_Trig(CLK := Reset);

// 무장(SET): 파이버 센서 100ms 연속 ON = 유효 케이스 (RESET 은 push 성공 시)
IF Valid_TON.Q THEN
    Case_Armed := TRUE;
END_IF

// 하강엣지 순간 후단 위치 캡처 (디바운스 통과 시 이 위치를 push — push 는 OFF_DEBOUNCE 만큼 늦어도 위치는 진짜 후단)
IF Fiber_Trig.Q THEN
    Trailing_Pos := Real_Position;
END_IF

// ===== 후단 확정(OFF_DEBOUNCE 연속 OFF) 시 기준점을 큐에 push =====
// OFF_DEBOUNCE 미만의 마진 OFF/블립은 Off_TON 이 리셋되어 무시 → 가까운 부품 조기 트리거 방지.
IF Auto_Mode AND Off_Confirm.Q AND Case_Armed THEN
    // push 성공 시에만 무장 해제. 큐 만재(거부)면 Case_Armed 유지 → 무음 유실 방지
    IF Queue.Push(Trailing_Pos) THEN
        Case_Armed := FALSE;
    END_IF
END_IF

// ===== head 기준점 + Trigger_Length 도달 시 1회 발동 + pop =====
bDistReached := FALSE;
IF Auto_Mode
   AND Trigger_Length > 0       // 길이 오설정(0/음수) 시 과트리거 방지(pop 보호)
   AND Queue.Count > 0
   AND NOT Trig_Pulse.Q         // ★ 직전 트리거 펄스(0.1s) 진행 중엔 발동 보류.
                                //   안 그러면 펄스폭 안에 들어온 다음 부품이 pop 되며 Trig_Position 만 덮어쓰고
                                //   카메라는 안 찍히는 desync(=가까운 부품 트리거거리 부정확) 발생.
   AND (Queue.HeadValue + Trigger_Length <= Real_Position) THEN
    bDistReached := TRUE;
    Trig_Position := Real_Position;   // 실제 발동 순간 엔코더 래치 — 카메라 실촬영 위치와 1:1 일치
    Queue.Pop();
END_IF

// 0.1s 펄스 정형
Trig_Pulse(IN := bDistReached, PT := T#0.1S);
Trigger := Trig_Pulse.Q;

// ===== 큐 flush =====
//  (1) 오토 이탈 / 컨베이어 역방향(Conveyor_CCW)
//  (2) 위치 불연속(엔코더 리셋 Set_Pos · 대형 역행 점프): head 기준점이 영구 도달불가가 되어
//      pop 정지 → stale 큐(Cam_Trig_Position 오류) 방지. 정상 전진/pop 시 Real 은 뒤로
//      점프하지 않으므로 오검출 없음. (RESET_JUMP_MIN 은 1스캔 최대 이송보다 크게 튜닝)
IF NOT Auto_Mode
   OR Conveyor_CCW
   OR ((Last_Real_Position - Real_Position) > RESET_JUMP_MIN) THEN
    Queue.Clear();
    Case_Armed := FALSE;
END_IF
Last_Real_Position := Real_Position;

// ===== 시스템 초기화 / 사이클말 큐 비움 (구 Vision_ST run7 의 큐 clear) =====
IF Reset_Trig.Q THEN
    Queue.Clear();
    Case_Armed := FALSE;
END_IF

END_FUNCTION_BLOCK

// ---- POUs/FB_LRealRingQueue.TcPOU
(* LREAL 링버퍼(FIFO) — 순차 push/pop. 좌표/엔코더 위치 등 범용 사용. *)
FUNCTION_BLOCK FB_LRealRingQueue
VAR CONSTANT
	CAPACITY : INT := 5;          // 링버퍼 칸 수(고정)
END_VAR
VAR
	buf  : ARRAY[0..4] OF LREAL;  // 기준점 저장(크기 = CAPACITY)
	head : INT;                   // pop 위치(가장 오래된 항목)
	tail : INT;                   // push 위치(다음 빈 칸)
	cnt  : INT;                   // 적재 수
END_VAR

METHOD Push : BOOL
VAR_INPUT
	val : LREAL;
END_VAR
IF cnt >= CAPACITY THEN
	Push := FALSE;            // 가득 — 거부
	RETURN;
END_IF
buf[tail] := val;
tail := (tail + 1) MOD CAPACITY;
cnt  := cnt + 1;
Push := TRUE;
END_METHOD

METHOD Pop : BOOL
IF cnt <= 0 THEN
	Pop := FALSE;            // 비어있음
	RETURN;
END_IF
head := (head + 1) MOD CAPACITY;
cnt  := cnt - 1;
Pop := TRUE;
END_METHOD

METHOD Clear
head := 0;
tail := 0;
cnt  := 0;
END_METHOD

PROPERTY Count : INT
GET
Count := cnt;
END_GET
END_PROPERTY

PROPERTY HeadValue : LREAL
GET
IF cnt > 0 THEN
	HeadValue := buf[head];
ELSE
	HeadValue := 0;
END_IF
END_GET
END_PROPERTY

END_FUNCTION_BLOCK

// ---- POUs/Vision/Move_Command.TcPOU
PROGRAM Move_Command
VAR
	Motor_Move_Trig          : R_TRIG;
	Move_Watchdog            : TON;

END_VAR



IF GVL_Calibration.Calibration_comp THEN
    GVL_Calibration.All_Motor_Wait_Pos_Moving := TRUE;  // (S) Set
END_IF


Motor_Move_Trig(CLK := GVL_Calibration.Motor_Move);

IF  Motor_Move_Trig.Q THEN
	GVL_Axis01.Calibration_Position := FALSE;
	GVL_Axis02.Calibration_Position := FALSE;
	GVL_Axis03.Calibration_Position := FALSE;
	GVL_Axis04.Calibration_Position := FALSE;
	GVL_Calibration.Calibration_Pos_Moving := TRUE;
END_IF

IF GVL_Axis01.Calibration_Position AND
   GVL_Axis02.Calibration_Position AND
   GVL_Axis03.Calibration_Position AND
   GVL_Axis04.Calibration_Position THEN
	GVL_Calibration.Motor_Move := FALSE;
	GVL_Calibration.Calibration_Pos_Moving := FALSE;
END_IF

// 잔류 해제 1: 이동을 지속할 수 없는 상태(모드 이탈/정지/세이프티)면 즉시 클리어
IF NOT GVL_System.Calibration_Mode OR GVL_System.Stop
   OR GVL_System.All_Motor_Stop OR NOT GVL_System.Safety_ALL_OK THEN
	GVL_Calibration.Motor_Move := FALSE;
	GVL_Calibration.Calibration_Pos_Moving := FALSE;
END_IF

// 잔류 해제 2: 워치독 — 이동 중 10초 초과 시 강제 클리어 (축 알람 등으로 완료 불가 케이스)
Move_Watchdog(IN := GVL_Calibration.Calibration_Pos_Moving, PT := T#10S);
IF Move_Watchdog.Q THEN
	GVL_Calibration.Motor_Move := FALSE;
	GVL_Calibration.Calibration_Pos_Moving := FALSE;
END_IF

END_PROGRAM

// ---- POUs/Work/Motion_Step_ST.TcPOU
PROGRAM Motion_Step_ST
VAR
    Vision_OK_Trig     : R_TRIG;             // 비전 OK 상승엣지(결과 캡처)
    VisionQueue        : FB_VisionDataQueue; // 비전 결과 큐(덮어쓰기 방지, 용량5)
    Vis_Item           : ST_VisionData;      // 큐 push 용 스크래치
    Vis_Head           : ST_VisionData;      // 큐 pop(Head) 용 스크래치
    Cam_Trig_Pos_Buf   : LREAL;              // 소비된 부품의 캠트리거 위치(Target X 보정 기준)
    Active_ID          : DINT;               // 현재 처리(압입) 중 부품의 비전 인식 ID
    Skip_Event         : BOOL;               // 이번 스캔 프레스 실패(skip) 발생 — NG 부저 트리거(매 스캔 클리어)
    NG_Playing         : BOOL;               // NG 모스 부저 재생 중
    NG_Timer           : TON;                // NG 패턴 경과시간 타이머(한 번 ≈ 1초)
    Cand_Target_X      : LREAL;              // pop 후보 부품의 현재 Target X (도달성 판단)
    Data_Initial       : BOOL;               // 캡처 직후 Data_Read/Vision_OK 초기화 예약
    Vision_Copy_Status : BOOL;               // 비전 캡처 게이트(오토 전용: Auto AND Safety)
    Stop_Req           : BOOL;               // (옵션) 프레스 실패 정지 요청 래치 — No=0(안전·X기어해제)에서 All_Motor_Stop 적용
    Auto_Resume_Trig   : R_TRIG;             // 오토 재요청 상승엣지(정지 해제·복구)
    X_Coupled          : BOOL;               // X(Axis02) 기어 커플 상태 추적 — Press_Start에서 래치, Work_End_Position에서 해제
    Manual_Nudge       : BOOL;               // 림보(Auto·Manual 둘다 OFF) 탈출용 수동요청 넛지 플래그
    Z_Torque_Timer      : TON;               // 압입 토크 임계 도달 지속 확인(하강 가속 스파이크 오검출 방지)
    Z_Stop_Timer        : TON;               // 토크완료 후 Z MC_Stop 정지 확인 디바운스
    // 디바운스 값(토크 도달 지속·정지 판정 속도·정지 확정 지속)은 GVL_Axis04 의 PERSISTENT 심볼로
    // 이관 → HMI/대시보드(ADS)에서 조절. 시간(ms UDINT)은 UDINT_TO_TIME 으로 TON.PT 에 전달.
END_VAR

// 엣지 검출 (매 스캔)
Vision_OK_Trig(CLK := GVL_Vision.Vision_OK);

// 코일 초기화
GVL_Motion_Step.Motion_Start := FALSE;
GVL_Motion_Step.Target_Pos_Moving := FALSE;
GVL_Motion_Step.Axis02_Work_Wait := FALSE;
GVL_Motion_Step.Press_Start := FALSE;
GVL_Motion_Step.Z_Press_Start := FALSE;
GVL_Motion_Step.Axis04_Wait_Pos_Moving := FALSE;
GVL_Motion_Step.Axis02_Stop := FALSE;
GVL_Motion_Step.All_Axis_Wait_Pos_Moving := FALSE;
GVL_Motion_Step.Work_Comp_Target_Pos_Moving := FALSE;
GVL_Motion_Step.All_Initial := FALSE;
Skip_Event := FALSE;   // 매 스캔 클리어 (skip 발생 스캔만 TRUE)

// ===== 비전 결과 캡처 (덮어쓰기 방지) =====
// 모션 가능여부와 무관하게, 가깝게 들어온 Vision_OK 결과를 매 엣지마다 큐에 전부 적재.
IF GVL_System.Auto_Mode AND Vision_OK_Trig.Q THEN
    Vis_Item.ID                := GVL_Vision.Data_Read_ID;        // 인식 ID 스냅샷
    Vis_Item.X                 := GVL_Vision.Data_Read_X;
    Vis_Item.Y                 := GVL_Vision.Data_Read_Y;
    Vis_Item.Rot               := GVL_Vision.Data_Read_R;
    Vis_Item.Cam_Trig_Position := GVL_Vision.Cam_Trig_Position;   // 캡처 시점 캠트리거 위치 스냅샷
    IF VisionQueue.Push(Vis_Item) THEN
        GVL_Vision.Vision_Q_Overflow := FALSE;
    ELSE
        GVL_Vision.Vision_Q_Overflow := TRUE;   // 큐 만재 → 무음 유실 방지 경보(용량↑ 또는 프레스 처리율↑)
        // 큐 만재로 미적재 → skip 보고 (reason 3)
        GVL_Vision.Skipped_ID_Buf[GVL_Vision.Skip_Count MOD 256]     := Vis_Item.ID;
        GVL_Vision.Skipped_Reason_Buf[GVL_Vision.Skip_Count MOD 256] := 3;
        GVL_Vision.Skip_Count := GVL_Vision.Skip_Count + 1;
        Skip_Event := TRUE;   // 프레스 실패 → 부저 펄스 트리거
    END_IF
    Data_Initial := TRUE;   // Data_Read/Vision_OK 초기화 → 다음 결과 수신 준비
END_IF

GVL_Vision.Vision_Q_Count := VisionQueue.Count;   // HMI 모니터

// ===== 비전 큐 flush (pop 보호: stale 항목 영구잔류 방지) =====
// 오토 이탈 / 시스템 초기화 시 큐 비움. (사이클말 No=40 에서는 비우지 않음 — 대기 부품 보존)
IF NOT GVL_System.Auto_Mode OR GVL_System.All_Initial THEN
    VisionQueue.Clear();
    GVL_Vision.Vision_Q_Overflow := FALSE;
END_IF

// ===== 모션 시퀀스 (CASE: 스캔당 1스텝만 — 같은 스캔 cascade/stale 판정 방지) =====
IF GVL_System.Auto_Mode THEN

    // Target X 위치 계산 (스텝이 읽기 전, No<>0 일 때 매 스캔 갱신)
    IF GVL_Motion_Step.No <> 0 THEN
        GVL_Vision.Target_X_Real_Position_Data := GVL_Vision.Data_Buffer_X - (GVL_Encoder.Real_Position - Cam_Trig_Pos_Buf);
    END_IF

    CASE GVL_Motion_Step.No OF

        0:  // 큐에서 다음 부품 pop. Wait 위치를 지나친(도달불가) 부품은 폐기(실패), 도달 가능한 것만 적재.
            IF Stop_Req THEN
                // (옵션) 실패 정지 요청 대기 — 사이클 안전종료·X 기어해제 유휴에서만 정지 적용. pop 보류.
                GVL_System.All_Motor_Stop := TRUE;     // Auto 차단(→ 수동, 아래 넛지가 Manual 진입)
                GVL_Conv.Motor_STOP := TRUE;           // 실제 컨베이어 정지(Conv.TcPOU 가 모든 컨베이어 출력 OFF)
            ELSIF VisionQueue.Count > 0 THEN
                Vis_Head := VisionQueue.HeadData;    // 가장 오래된 항목
                Cand_Target_X := Vis_Head.X - (GVL_Encoder.Real_Position - Vis_Head.Cam_Trig_Position);
                IF Cand_Target_X >= GVL_Axis02.Wait_Position_Data THEN
                    // 아직 Wait 전 → 도달 가능 → 적재 + 시작
                    VisionQueue.Pop();
                    GVL_Vision.Data_Buffer_X := Vis_Head.X;
                    GVL_Vision.Data_Buffer_Y := Vis_Head.Y;
                    GVL_Vision.Data_Buffer_R := Vis_Head.Rot;
                    Cam_Trig_Pos_Buf         := Vis_Head.Cam_Trig_Position;
                    Active_ID                := Vis_Head.ID;     // 처리 중 부품 ID 보관(압입 시 보고)
                    GVL_Motion_Step.Motion_Start := TRUE; // not use
                    GVL_Motion_Step.No := 1;
                ELSE
                    // Wait 통과(이미 지나침, 도달불가) → 폐기 + skip 보고 (reason 1)
                    GVL_Vision.Skipped_ID_Buf[GVL_Vision.Skip_Count MOD 256]     := Vis_Head.ID;
                    GVL_Vision.Skipped_Reason_Buf[GVL_Vision.Skip_Count MOD 256] := 1;
                    GVL_Vision.Skip_Count := GVL_Vision.Skip_Count + 1;
                    Skip_Event := TRUE;   // 프레스 실패 → 부저 펄스 트리거
                    VisionQueue.Pop();   // 폐기, 다음 부품 시도
                END_IF
            END_IF

        1:  // R/Y 타겟 이동 시작 (블로킹 안 함 — 대기/sync 구간 병렬 이동, Z 프레스 직전 도달 확인)
            GVL_Motion_Step.Target_Pos_Moving := TRUE; // reference axis03_auto, axis01_auto
            GVL_Motion_Step.No := 5;

        5:  // Axis02 Work Wait (R/Y 병렬 이동 지속)
            GVL_Motion_Step.Target_Pos_Moving := TRUE;   // R/Y 계속 타겟으로
            GVL_Motion_Step.Axis02_Work_Wait := TRUE;
            IF GVL_Vision.Target_X_Real_Position_Data <= GVL_Axis02.Wait_Position_Data THEN
                GVL_Motion_Step.No := 10;
            END_IF

        10: // Press Start (sync). R/Y 타겟 도달 후에만 Z 프레스. R/Y 지연으로 압입범위 지나치면 실패 복귀.
            GVL_Motion_Step.Target_Pos_Moving := TRUE;   // R/Y 타겟 유지(sync 구간 병렬 이동)
            GVL_Motion_Step.Press_Start := TRUE;
            IF GVL_Vision.Target_X_Real_Position_Data <= (GVL_Axis02.Wait_Position_Data - GVL_Axis02.Sync_Data)
               AND GVL_Axis03.Target_Position AND GVL_Axis01.Target_Position THEN
                GVL_Motion_Step.Z_Press_Start := TRUE;
            END_IF

            // ===== 토크 압입 완료 판정 =====
            // 실제토크(GVL_Axis04.Torque_Actual, PDO)가 임계값(Press_Torque_Reach_Data) 이상으로
            // Press_Torque_Reach_Time_Data(ms) 지속되면(가속 스파이크 오검출 방지) 목표 위치 미도달이어도 토크한계 도달로 완료.
            Z_Torque_Timer(IN := GVL_Motion_Step.Z_Press_Start
                                 AND ABS(GVL_Axis04.Torque_Actual) >= GVL_Axis04.Press_Torque_Reach_Data
                                 AND NOT GVL_Axis04.Work_End_Position,
                           PT := UDINT_TO_TIME(GVL_Axis04.Press_Torque_Reach_Time_Data));

            IF GVL_Axis04.Work_End_Position THEN
                // 정상(위치도달) 완료 — 기존 경로. 무손실 압입 ID 보고: 현재 count 슬롯에 ID 기록 → count 증가
                GVL_Vision.Pressed_ID_Buf[GVL_Vision.Press_Count MOD 256] := Active_ID;
                GVL_Vision.Press_Count := GVL_Vision.Press_Count + 1;   // vision은 Press_Count 증가분만큼 Buf 읽음
                GVL_Motion_Step.No := 20;
            ELSIF Z_Torque_Timer.Q THEN
                // 토크한계 도달 완료 — 위치 미도달(눌러박힘)이라 press MoveAbsolute 를 MC_Stop 으로 끊어야 함(No=15).
                // 컨베이어/부품 눌러박힘으로 Work_End_Position 이 안 떠 No=10 에 머물며 계속 누르던 hang 방지.
                GVL_Vision.Pressed_ID_Buf[GVL_Vision.Press_Count MOD 256] := Active_ID;
                GVL_Vision.Press_Count := GVL_Vision.Press_Count + 1;
                GVL_Motion_Step.No := 15;
            ELSIF GVL_Vision.Target_X_Real_Position_Data < 0
                  AND NOT GVL_Motion_Step.Z_Press_Start THEN
                // 미압입(R/Y 지연) abort → skip 보고 (reason 2)
                GVL_Vision.Skipped_ID_Buf[GVL_Vision.Skip_Count MOD 256]     := Active_ID;
                GVL_Vision.Skipped_Reason_Buf[GVL_Vision.Skip_Count MOD 256] := 2;
                GVL_Vision.Skip_Count := GVL_Vision.Skip_Count + 1;
                Skip_Event := TRUE;   // 프레스 실패 → 부저 펄스 트리거
                GVL_Motion_Step.No := 25;   // Z 미진입, 부품이 0(센서 닿기 전 한계) 지나침 → No=25 MC_Stop 복귀
            END_IF

        15: // 토크 압입 완료 후 Z 강제정지(MC_Stop) → 정지 확인 → 복귀(No=20)
            // press MoveAbsolute 는 Execute 를 떨궈도 안 멈추므로(계속 목표로 누름) Z MC_Stop(Axis04_Stop_01)로 확실히 끊는다.
            // GVL_Main_Step.Press_Stop → Axis04_Status 의 MC_Stop Execute(전용 훅). 정지 확인 후 해제해야 다음 복귀 move 가능.
            Z_Stop_Timer(IN := ABS(GVL_Axis04.Real_Velocity) < GVL_Axis04.Press_Stop_Vel_Data,
                         PT := UDINT_TO_TIME(GVL_Axis04.Press_Stop_Time_Data));
            IF Z_Stop_Timer.Q THEN
                GVL_Main_Step.Press_Stop := FALSE;   // MC_Stop 해제 → No=20 Wait 복귀 move 실행 가능
                GVL_Motion_Step.No := 20;
            ELSE
                GVL_Main_Step.Press_Stop := TRUE;    // Z MC_Stop 유지(press 정지)
            END_IF

        20: // Axis04 Wait Pos Moving
            IF GVL_Axis02.Real_Position <-1 THEN
                GVL_Motion_Step.Press_Start := FALSE;
                GVL_Motion_Step.Axis04_Wait_Pos_Moving := TRUE;
                GVL_Motion_Step.No := 25;
            END_IF
            IF GVL_Axis02.Real_Position <= (GVL_Axis02.Work_End_Position_Data + 10) THEN
                GVL_Motion_Step.Axis04_Wait_Pos_Moving := TRUE;
            END_IF
            IF GVL_Axis02.Real_Position <= GVL_Axis02.Work_End_Position_Data THEN
                GVL_Motion_Step.No := 25;
            END_IF

        25: // Axis02 Stop
            GVL_Motion_Step.Axis02_Stop := TRUE;
            IF GVL_Axis02.Work_End_Position THEN
                GVL_Motion_Step.No := 30;
            END_IF

        30: // All Axis Wait Pos Moving
            GVL_Motion_Step.All_Axis_Wait_Pos_Moving := TRUE;
            IF GVL_System.ALL_Wait_Position THEN
                GVL_Motion_Step.No := 40;
            END_IF

        40: // 사이클말 — All Initial + 버퍼/카피완료 초기화 (비전 큐는 비우지 않음: 대기 부품 보존)
            GVL_Motion_Step.All_Initial := TRUE;
            GVL_Vision.Data_Buffer_X := 0;
            GVL_Vision.Data_Buffer_Y := 0;
            GVL_Vision.Data_Buffer_R := 0;
            GVL_Vision.Target_X_Real_Position_Data := 0;
            GVL_Motion_Step.No := 0;

    ELSE
        GVL_Motion_Step.No := 0;   // 미정의 스텝값 → 안전 복귀(유휴)

    END_CASE

END_IF

// ===== X 기어 커플 추적 + Auto 이탈 시 강제 디커플 (수동전환·안전 등 어떤 이유로든 기어인 방치 방지) =====
// 기존엔 디커플 체인(Axis02_Stop→MC_Stop→MC_GearOut)이 Auto No=25 에서만 트리거 → Auto 빠지면 X 기어인 잔류.
// Press_Start(기어인)에서 커플 래치, Work_End_Position(MC_GearOut.Done)에서 해제.
IF GVL_Motion_Step.Press_Start THEN
    X_Coupled := TRUE;
END_IF
IF GVL_Axis02.Work_End_Position THEN
    X_Coupled := FALSE;
END_IF
// Auto 가 빠졌는데 X가 아직 커플이면 → No 머신과 무관하게 디커플 체인 강제 구동(Axis02_Command 는 매 스캔 실행).
// 디커플 완료 시 X_Coupled 해제 → 코일초기화로 Axis02_Stop 자동 release → 수동 조그 가능.
IF X_Coupled AND NOT GVL_System.Auto_Mode THEN
    GVL_Motion_Step.Axis02_Stop := TRUE;
END_IF

// ===== Z 정지훅(Press_Stop) 안전 해제 =====
// 토크완료 정지(No=15)용 Z MC_Stop 훅. 오토 이탈·초기화 시 래치 잔류로 Z가 정지에 물려 수동조작·복구를
// 방해하지 않도록 해제. (No=15 정상 진행 시엔 그 스텝에서 정지확인 후 스스로 해제)
IF NOT GVL_System.Auto_Mode OR GVL_System.All_Initial THEN
    GVL_Main_Step.Press_Stop := FALSE;
END_IF

// Vision 데이터 초기화 (캡처 직후 다음 결과 수신 준비) =====
IF Data_Initial OR GVL_System.All_Initial THEN
    GVL_Vision.Data_Read_X := 0;
    GVL_Vision.Data_Read_Y := 0;
    GVL_Vision.Data_Read_R := 0;
    GVL_Vision.Vision_OK := FALSE;
    Data_Initial := FALSE;
END_IF

// ===== 프레스 실패(비전 왔는데 미압입) 부저 — "NG" 모스부호 (N:―· G:――·), 알람부저와 구분 =====
// 단위 60ms, 한 번 재생 ≈ 1초. skip 시 1회 재생. 중지·에러 없이 부저만, System 부저에 OR(비파괴).
IF NG_Timer.Q THEN
    NG_Playing := FALSE;
END_IF
IF Skip_Event THEN
    NG_Playing := TRUE;   // 실패 → NG 재생 시작(재생 중 추가 실패는 현재 재생 끝난 뒤 새로 시작)
END_IF
NG_Timer(IN := NG_Playing, PT := T#1020MS);
GVL_System.Buzzer := GVL_System.Buzzer OR (NG_Playing AND (
       (NG_Timer.ET <  T#180MS)                                  // N: dash(―)
    OR (NG_Timer.ET >= T#240MS AND NG_Timer.ET < T#300MS)        // N: dot(·)
    OR (NG_Timer.ET >= T#480MS AND NG_Timer.ET < T#660MS)        // G: dash(―)
    OR (NG_Timer.ET >= T#720MS AND NG_Timer.ET < T#900MS)        // G: dash(―)
    OR (NG_Timer.ET >= T#960MS AND NG_Timer.ET < T#1020MS)));    // G: dot(·)

// ===== (옵션) 프레스 실패 시 컨베이어 정지 + 수동 전환 — vision 이 GVL_Vision.Stop_On_Fail 로 ON/OFF =====
// 실패(skip) → Stop_Req 래치. 실제 정지는 No=0(사이클 안전종료·X 기어해제)에서 All_Motor_Stop 적용(위 CASE 0).
// All_Motor_Stop=TRUE → Auto 차단(→ 수동, 넛지가 Manual 진입) / Motor_STOP=TRUE → 컨베이어 정지(Conv.TcPOU). 알람/에러 없음. 수동 조작은 안 막음.
// 복구: 오토 재요청(HMI_Auto_Mode) 상승엣지 또는 리셋(All_Initial) 시 Stop_Req·All_Motor_Stop·Motor_STOP 해제.
IF Skip_Event AND GVL_Vision.Stop_On_Fail THEN
    Stop_Req := TRUE;
END_IF
Auto_Resume_Trig(CLK := GVL_System.HMI_Auto_Mode);
IF Auto_Resume_Trig.Q OR GVL_System.All_Initial THEN
    Stop_Req := FALSE;
    GVL_System.All_Motor_Stop := FALSE;
    GVL_Conv.Motor_STOP := FALSE;
END_IF

// ===== 림보(Auto·Manual 둘 다 OFF) 자동 탈출 → 수동 진입 =====
// Manual_Mode 진입은 (HMI_Manual_Mode AND NOT Each_Motor_Busy) 게이트라, 동작 중(gear-in/압입) 모드전환 시
// Auto 자기유지만 끊겨 Auto OFF·Manual 못 들어가는 림보 발생(모멘터리 수동버튼·fail-stop 공통).
// 모터 정지·안전·오토요청 아님이면 수동요청을 넣어 Manual 을 래치시키고, 진입되면 떼어냄.
// (HMI 는 버튼 누를 때만 HMI_Manual_Mode 를 쓰므로 평소엔 건드리지 않아 충돌 없음)
IF NOT GVL_System.Auto_Mode AND NOT GVL_System.Manual_Mode
   AND GVL_System.Safety_ALL_OK AND NOT GVL_System.Each_Motor_Busy
   AND NOT GVL_System.HMI_Auto_Mode THEN
    GVL_System.HMI_Manual_Mode := TRUE;    // 수동 진입 넛지
    Manual_Nudge := TRUE;
ELSIF Manual_Nudge THEN
    GVL_System.HMI_Manual_Mode := FALSE;   // 넛지로 set 한 것만 해제(진입 완료 후) — 오토 복귀 막지 않게
    Manual_Nudge := FALSE;
END_IF

END_PROGRAM

// ---- POUs/FB_VisionDataQueue.TcPOU
(* 비전 결과(ST_VisionData) 링버퍼(FIFO) — 가깝게 연속 도착하는 결과를 덮어쓰지 않고 적재.
   FB_LRealRingQueue 와 동일한 링버퍼 패턴을 좌표 세트(struct)용으로 확장. *)
FUNCTION_BLOCK FB_VisionDataQueue
VAR CONSTANT
    CAPACITY : INT := 5;           // 링버퍼 칸 수(고정) — 버스트 폭에 맞춰 튜닝
END_VAR
VAR
    buf  : ARRAY[0..4] OF ST_VisionData;   // 결과 저장(크기 = CAPACITY)
    head : INT;                            // pop 위치(가장 오래된 항목)
    tail : INT;                            // push 위치(다음 빈 칸)
    cnt  : INT;                            // 적재 수
END_VAR

METHOD Push : BOOL
VAR_INPUT
    val : ST_VisionData;
END_VAR
IF cnt >= CAPACITY THEN
    Push := FALSE;            // 가득 — 거부(무음 유실 방지: 호출측에서 경보)
    RETURN;
END_IF
buf[tail] := val;
tail := (tail + 1) MOD CAPACITY;
cnt  := cnt + 1;
Push := TRUE;
END_METHOD

METHOD Pop : BOOL
IF cnt <= 0 THEN
    Pop := FALSE;            // 비어있음
    RETURN;
END_IF
head := (head + 1) MOD CAPACITY;
cnt  := cnt - 1;
Pop := TRUE;
END_METHOD

METHOD Clear
head := 0;
tail := 0;
cnt  := 0;
END_METHOD

PROPERTY Count : INT
GET
Count := cnt;
END_GET
END_PROPERTY

PROPERTY HeadData : ST_VisionData
GET
IF cnt > 0 THEN
    HeadData := buf[head];
END_IF
END_GET
END_PROPERTY

END_FUNCTION_BLOCK

// ---- POUs/Vision/Mastering.TcPOU
PROGRAM Mastering
VAR
	Move_Margin : LREAL;            // 목표 복귀거리 (mastering_vision_x - Axis02 대기위치), STEP20 진입 시 래치
	Start_Position : LREAL;         // 마스터링 시작 기준 위치
	Sensor_Position : LREAL;        // 비전 시작 센서 감지 위치
	Forward_Distance : LREAL;       // 시작점 기준 정방향 이동거리
	Shot_Position : LREAL;          // 정방향 카메라 촬영 위치
	Back_Distance : LREAL;          // Back 단계 이동량 (대기위치 기준 CCW 복귀량)
	Back_Start_Position : LREAL;    // Back 단계 시작(대기) 시점의 컨베이어 위치
	Fiber_Sensor_Trig  : R_TRIG;
	Back_Pos_Trig : R_TRIG;

	Mastering_Step : INT;

	fbCamPulse : TP;
	bCamTrigTP : BOOL;
	Settle_Timer : TON;             // STEP20 재촬영 전 정지·정착 대기 타이머

END_VAR


Fiber_Sensor_Trig(CLK := GVL_System.Fiber_Sensor);
Back_Pos_Trig(CLK := GVL_Mastering.Back_Trig);

fbCamPulse(IN := bCamTrigTP, PT := T#200MS);
bCamTrigTP := FALSE;

// 마스터링(수동) 모드에서 카메라 물리 트리거(GVL_Vision.Cam_Trigger) 구동.
// 오토모드는 Vision_ST 가 구동 — 모드가 배타적이라 두 POU 가 같은 출력을 안 다툼.
IF GVL_System.Manual_Mode THEN
    GVL_Vision.Cam_Trigger := fbCamPulse.Q;
END_IF


(* ──────────────────────────────────────────────────────────────
   [Back 트리거 처리]
   Back 트리거 상승 엣지 발생 시 현재 엔코더 위치를 Back_Shot_Position에 저장
   ────────────────────────────────────────────────────────────── *)
IF Back_Pos_Trig.Q THEN
    GVL_Mastering.Back_Shot_Position := GVL_Encoder.Real_Position;
END_IF


(* ==============================================================
   [초기화 처리] All_Initial + Manual_Mode 조건에서 전체 변수 리셋
   ============================================================== *)
IF GVL_System.All_Initial AND GVL_System.Manual_Mode THEN

    (* 내부 연산 변수 초기화 *)
    Start_Position      := 0;
    Sensor_Position     := 0;
    Forward_Distance    := 0;
    Shot_Position       := 0;
    Back_Distance       := 0;

    (* GVL 마스터링 변수 초기화 *)
    GVL_Mastering.mastering_vision_x      := 0;
    GVL_Mastering.Case_Length_Check_Start := FALSE;
    GVL_Mastering.Back_Trig               := FALSE;
    GVL_Mastering.Case_Length             := 0;

    (* 스텝 초기화 *)
    Mastering_Step                        := 0;

END_IF


(* ==============================================================
   [마스터링 메인 시퀀스] Case_Length_Check_Start = TRUE 조건에서 실행
   ============================================================== *)
IF GVL_Mastering.Case_Length_Check_Start AND GVL_System.Manual_Mode THEN


    (* ── STEP 0 : 마스터링 시작 초기화 및 컨베이어 역방향 구동 ── *)
    IF  Mastering_Step = 0 THEN

        (* 내부 변수 초기화 *)
        Sensor_Position     := 0;
        Forward_Distance    := 0;
        Shot_Position       := 0;
        Back_Distance       := 0;
        Settle_Timer(IN := FALSE, PT := T#2S);   (* 정착 타이머 리셋 *)

        (* GVL 마스터링 변수 초기화 *)
        GVL_Mastering.mastering_vision_x  := 0;
        GVL_Mastering.Back_Trig           := FALSE;
        GVL_Mastering.Case_Length         := 0;

        (* 케이스 시작 위치 기록 후 컨베이어 역방향(CCW) 저속 구동 시작 *)
        Start_Position := GVL_Encoder.Real_Position;

        GVL_Conv.HMI_Motor_CCW       := TRUE;
        GVL_Conv.HMI_Motor_Low_Speed := TRUE;

        Mastering_Step := 5;

    END_IF


    (* ── STEP 5 : 비전 시작 센서 감지 → 케이스 길이 계산 ── *)
    IF Fiber_Sensor_Trig.Q AND Mastering_Step = 5 THEN

        (* 센서 감지 시점의 엔코더 위치 저장 → 케이스 길이 계산 *)
        Sensor_Position              := GVL_Encoder.Real_Position;
        GVL_Conv.HMI_Motor_CCW       := FALSE;
        GVL_Conv.HMI_Motor_Low_Speed := FALSE;

        GVL_Mastering.Case_Length := Start_Position - Sensor_Position;

        (* 케이스 길이가 유효할 때만 다음 스텝으로 진행 *)
        IF GVL_Mastering.Case_Length <> 0 THEN
            Mastering_Step := 10;
        END_IF

    END_IF


    (* ── STEP 10 : 컨베이어 정방향 구동 + 카메라 트리거 위치 탐색 ── *)
    IF GVL_Mastering.Case_Length <> 0 AND Mastering_Step = 10 THEN

        (* 컨베이어 정방향(CW) 저속 구동 *)
        GVL_Conv.HMI_Motor_CW        := TRUE;
        GVL_Conv.HMI_Motor_Low_Speed := TRUE;

        (* 현재 이동 거리 갱신 (기준위치 Start_Position 기준) *)
        Forward_Distance := GVL_Encoder.Real_Position - Start_Position;

        IF Forward_Distance >= 0 THEN

            (* 카메라 트리거 활성화 및 촬영 위치 저장 *)
            bCamTrigTP    := TRUE;
            Shot_Position := GVL_Encoder.Real_Position;

            (* 카메라 실제 트리거 신호 수신 시 다음 스텝으로 진행 *)
            IF GVL_Vision.Cam_Trigger AND Shot_Position <> 0 THEN
                Mastering_Step := 15;
            END_IF

        END_IF

    END_IF


    (* ── STEP 15 : 비전 결과 수신 대기 + 정지 조건 판단 ── *)
    IF Mastering_Step = 15 THEN

        (* 비전 결과 수신 완료 시 정지 *)
        IF GVL_Mastering.mastering_vision_x <> 0 THEN
            GVL_Conv.HMI_Motor_CW         := FALSE;
            GVL_Conv.HMI_Motor_Low_Speed  := FALSE;
            GVL_Conv.Conv_Motor_CW        := FALSE;
            GVL_Conv.Conv_Motor_Low_Speed := FALSE;
            (* Back 복귀 기준점(대기위치)과 목표 복귀거리(Move_Margin)를 진입 시점에 래치 *)
            Back_Start_Position := GVL_Encoder.Real_Position;
            Move_Margin         := GVL_Mastering.mastering_vision_x - GVL_Axis02.Wait_Position_Data;
            Mastering_Step := 20;
        END_IF

    END_IF


    (* ── STEP 20 : Axis04 마스터링 위치 이동 → 역방향 재촬영 ── *)
    IF Mastering_Step = 20 AND GVL_Mastering.Back_Trig THEN

        (* Axis04를 마스터링 위치로 이동 명령 *)
        GVL_Axis04.M_Mastering_Pos_Move := TRUE;

        IF GVL_Axis04.Mastering_Position THEN

            (* 대기위치(Back 시작점) 대비 역방향(CCW=엔코더 감소) 복귀 이동량 계산 *)
            Back_Distance := Back_Start_Position - GVL_Encoder.Real_Position;

            IF Back_Distance < Move_Margin THEN

                (* 목표 미도달 → 컨베이어 역방향(CCW) 저속 복귀 주행 *)
                GVL_Conv.HMI_Motor_CCW       := TRUE;
                GVL_Conv.HMI_Motor_Low_Speed := TRUE;

            ELSE

                (* 목표(Move_Margin) 도달 → 컨베이어 정지 *)
                GVL_Conv.HMI_Motor_CCW        := FALSE;
                GVL_Conv.HMI_Motor_Low_Speed  := FALSE;
                GVL_Conv.Conv_Motor_CCW       := FALSE;
                GVL_Conv.Conv_Motor_Low_Speed := FALSE;

                (* 정지·정착 대기 2초 (제동/관성 정착 + 모션블러 제거) *)
                Settle_Timer(IN := TRUE, PT := T#2S);

                (* 정착 완료 후 카메라 트리거 → 노출=래치=정지위치 일치 *)
                IF Settle_Timer.Q THEN

                    bCamTrigTP := TRUE;

                    IF fbCamPulse.Q AND GVL_Vision.Cam_Trigger THEN
                        GVL_Mastering.Reshot_Position   := GVL_Encoder.Real_Position;
                        GVL_Axis04.M_Mastering_Pos_Move := FALSE;
                        Mastering_Step := 25;
                    END_IF

                END_IF

            END_IF

        END_IF

    END_IF

    (* ── STEP 25 : 마스터링 완료 처리 ── *)
    IF Mastering_Step = 25 THEN

        (* 마스터링 관련 플래그 및 스텝 초기화 → 시퀀스 종료 *)
        GVL_Mastering.Case_Length_Check_Start := FALSE;
        GVL_Mastering.Back_Trig               := FALSE;
        Mastering_Step                        := 0;

    END_IF


END_IF  (* Case_Length_Check_Start *)

END_PROGRAM

// ---- POUs/Work/GOST.TcPOU
PROGRAM GOST
VAR
	all_work_end : BOOL;
	ton01 : TON;
END_VAR

all_work_end := GVL_Axis01.Work_End_Position AND GVL_Axis02.Work_End_Position AND GVL_Axis03.Work_End_Position AND GVL_Axis04.Work_End_Position;
TON01(IN := GVL_System.ALL_Wait_Position , PT := T#200MS);
IF GVL_System.GOST_MODE AND GVL_System.ALL_Wait_Position AND TON01.Q THEN
	GVL_Axis01.M_Work_End_Pos_Move := TRUE;
	GVL_Axis02.M_Work_End_Pos_Move := TRUE;
	GVL_Axis03.M_Work_End_Pos_Move := TRUE;	
	GVL_Axis04.M_Work_End_Pos_Move := TRUE;
	
	
END_IF

IF all_work_end AND GVL_System.GOST_MODE THEN
		GVL_Axis01.M_Wait_Pos_Move := TRUE;
		GVL_Axis02.M_Wait_Pos_Move := TRUE;
		GVL_Axis03.M_Wait_Pos_Move := TRUE;	
		GVL_Axis04.M_Wait_Pos_Move := TRUE;
	END_IF

END_PROGRAM

// ---- POUs/Axis01_R/Axis01_Interlock_ST.TcPOU
PROGRAM Axis01_Interlock_ST
VAR
    Always_ON      : BOOL := TRUE;
    Always_OFF     : BOOL := FALSE;
    Axis02_Safe    : BOOL;
    InRange_Home   : BOOL;
    InRange_Wait   : BOOL;
    InRange_Target : BOOL;
    InRange_Work   : BOOL;
END_VAR

VAR CONSTANT
    AXIS02_SAFE_LIMIT : REAL := 55.0;
    R_MIN             : REAL := -10.0;
    R_MAX             : REAL := 10.0;
END_VAR

END_PROGRAM

// ---- POUs/Axis02_X/Axis02_Interlock_ST.TcPOU
PROGRAM Axis02_Interlock_ST
VAR
//System_Bit
	Always_ON	:	BOOL	:=TRUE	;//상시 ON 
	Always_OFF	:	BOOL	:=FALSE	;//상시 OFF
	AxisRangeOK      : BOOL;
    AxisRangeOK_NoZ  : BOOL;  // Axis04 없는 버전
	YOK: BOOL;
	ROK: BOOL;
	ZOK: BOOL;
END_VAR

VAR CONSTANT
    AXIS02_SAFE_LIMIT : REAL := 55.0;
END_VAR

END_PROGRAM

// ---- POUs/Axis03_Y/Axis03_Interlock_ST.TcPOU
PROGRAM Axis03_Interlock_ST
VAR
    Always_ON    : BOOL := TRUE;
    Always_OFF   : BOOL := FALSE;
    Axis02_Safe  : BOOL;
    InRange_Home : BOOL;
    InRange_Wait : BOOL;
    InRange_Work : BOOL;
END_VAR

VAR CONSTANT
    AXIS02_SAFE_LIMIT : REAL := 55.0;
    Y_MIN             : REAL := -24;
    Y_MAX             : REAL := 24;
END_VAR

END_PROGRAM

// ---- POUs/Axis04_Z/Axis04_Set_Work_End_Speed.TcPOU
PROGRAM Axis04_Set_Work_End_Speed
VAR
END_VAR


IF GVL_System.Manual_Mode THEN 
	GVL_Axis04.Work_End_Speed := 30 ;
ELSE 
	GVL_Axis04.Work_End_Speed:= 100;
END_IF

END_PROGRAM

// ---- POUs/System/Login_Timer.TcPOU
PROGRAM Login_Timer
VAR_INPUT
	tLoginTimer : TON;	
END_VAR

(* 로그인 상태에서 타이머 동작 *)
IF GVL_System.Login THEN 
	GVL_System.LoginLamp := TRUE;	
END_IF

tLoginTimer(
    IN := GVL_System.LoginLamp,
    PT := T#30m
);

(* 30분 경과 시 자동 로그아웃 *)
IF tLoginTimer.Q THEN
    GVL_System.LoginLamp := FALSE;
END_IF

END_PROGRAM
